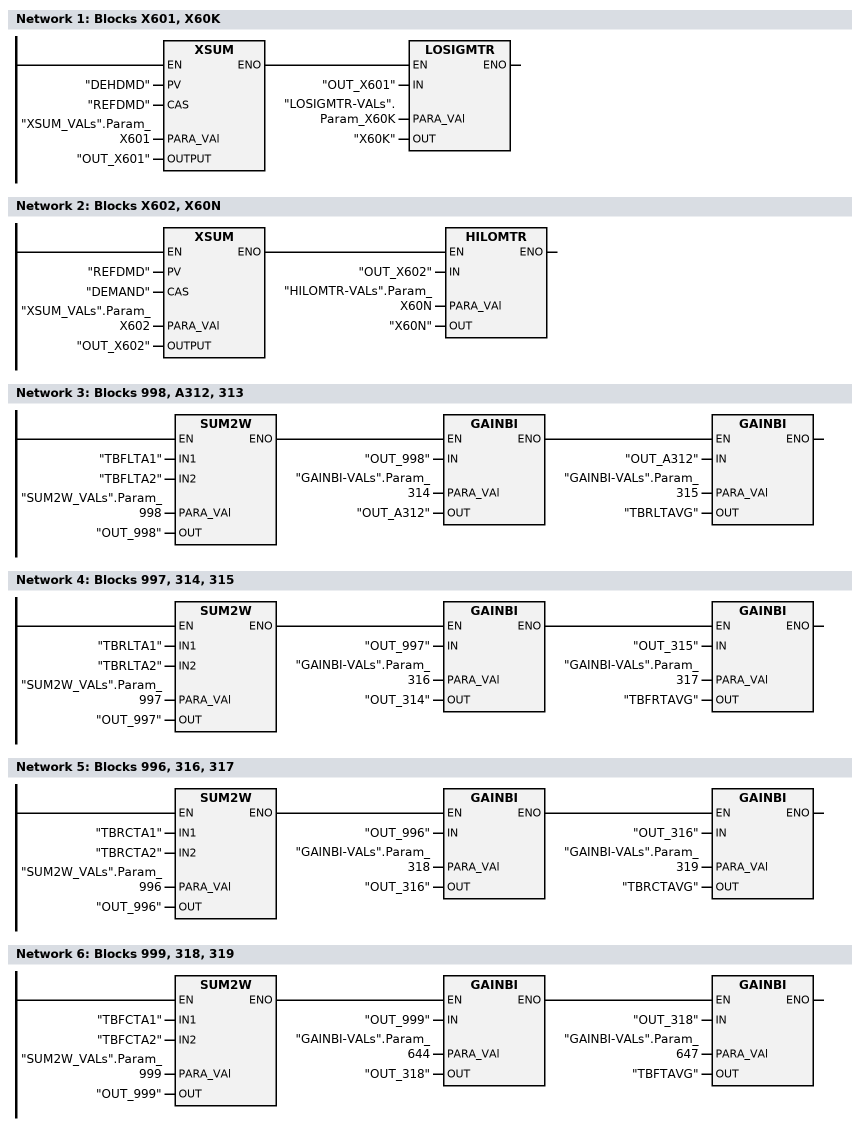
NETWORK
TITLE = Blocks X601, X60K
      A(;
      CALL  "XSUM" (
           PV                       := "DEHDMD",
           CAS                      := "REFDMD",
           PARA_VAl                 := "XSUM_VALs".Param_X601,
           OUTPUT                   := "OUT_X601");
      A     BR;
      );
      JNB   _001;
      CALL  "LOSIGMTR" (
           IN                       := "OUT_X601",
           PARA_VAl                 := "LOSIGMTR-VALs".Param_X60K,
           OUT                      := "X60K");
_001: NOP   0;
NETWORK
TITLE = Blocks X602, X60N
      A(;
      CALL  "XSUM" (
           PV                       := "REFDMD",
           CAS                      := "DEMAND",
           PARA_VAl                 := "XSUM_VALs".Param_X602,
           OUTPUT                   := "OUT_X602");
      A     BR;
      );
      JNB   _002;
      CALL  "HILOMTR" (
           IN                       := "OUT_X602",
           PARA_VAl                 := "HILOMTR-VALs".Param_X60N,
           OUT                      := "X60N");
_002: NOP   0;
NETWORK
TITLE = Blocks 998, A312, 313
      A(;
      A(;
      CALL  "SUM2W" (
           IN1                      := "TBFLTA1",
           IN2                      := "TBFLTA2",
           PARA_VAl                 := "SUM2W_VALs".Param_998,
           OUT                      := "OUT_998");
      A     BR;
      );
      JNB   _003;
      CALL  "GAINBI" (
           IN                       := "OUT_998",
           PARA_VAl                 := "GAINBI-VALs".Param_314,
           OUT                      := "OUT_A312");
_003: A     BR;
      );
      JNB   _004;
      CALL  "GAINBI" (
           IN                       := "OUT_A312",
           PARA_VAl                 := "GAINBI-VALs".Param_315,
           OUT                      := "TBRLTAVG");
_004: NOP   0;
NETWORK
TITLE = Blocks 997, 314, 315
      A(;
      A(;
      CALL  "SUM2W" (
           IN1                      := "TBRLTA1",
           IN2                      := "TBRLTA2",
           PARA_VAl                 := "SUM2W_VALs".Param_997,
           OUT                      := "OUT_997");
      A     BR;
      );
      JNB   _005;
      CALL  "GAINBI" (
           IN                       := "OUT_997",
           PARA_VAl                 := "GAINBI-VALs".Param_316,
           OUT                      := "OUT_314");
_005: A     BR;
      );
      JNB   _006;
      CALL  "GAINBI" (
           IN                       := "OUT_315",
           PARA_VAl                 := "GAINBI-VALs".Param_317,
           OUT                      := "TBFRTAVG");
_006: NOP   0;
NETWORK
TITLE = Blocks 996, 316, 317
      A(;
      A(;
      CALL  "SUM2W" (
           IN1                      := "TBRCTA1",
           IN2                      := "TBRCTA2",
           PARA_VAl                 := "SUM2W_VALs".Param_996,
           OUT                      := "OUT_996");
      A     BR;
      );
      JNB   _007;
      CALL  "GAINBI" (
           IN                       := "OUT_996",
           PARA_VAl                 := "GAINBI-VALs".Param_318,
           OUT                      := "OUT_316");
_007: A     BR;
      );
      JNB   _008;
      CALL  "GAINBI" (
           IN                       := "OUT_316",
           PARA_VAl                 := "GAINBI-VALs".Param_319,
           OUT                      := "TBRCTAVG");
_008: NOP   0;
NETWORK
TITLE = Blocks 999, 318, 319
      A(;
      A(;
      CALL  "SUM2W" (
           IN1                      := "TBFCTA1",
           IN2                      := "TBFCTA2",
           PARA_VAl                 := "SUM2W_VALs".Param_999,
           OUT                      := "OUT_999");
      A     BR;
      );
      JNB   _009;
      CALL  "GAINBI" (
           IN                       := "OUT_999",
           PARA_VAl                 := "GAINBI-VALs".Param_644,
           OUT                      := "OUT_318");
_009: A     BR;
      );
      JNB   _00a;
      CALL  "GAINBI" (
           IN                       := "OUT_318",
           PARA_VAl                 := "GAINBI-VALs".Param_647,
           OUT                      := "TBFTAVG");
_00a: NOP   0;
NETWORK
TITLE = Blocks AIN, 311, X222, X22M
      A(;
      A     "X01I";
      =     L 0.0;
      BLD   103;
      A(;
      A(;
      CALL  "AIN" , "AIN_VALs_POS_2" (
           IN                       := "ROTECC_W",
           OUT                      := "ROTECC");
      A     BR;
      );
      JNB   _00b;
      CALL  "GAINBI" (
           IN                       := "ROTECC",
           PARA_VAl                 := "GAINBI-VALs".Param_313,
           OUT                      := "ROTECCE");
_00b: A     BR;
      );
      JNB   _00c;
      CALL  "TRANSF" (
           FLAG                     := L 0.0,
           IN1_y                    := "A50",
           IN2_n                    := "ROTECCE",
           OUT                      := "OUT_X222");
_00c: A     BR;
      );
      JNB   _00d;
      CALL  "HISIGMTR" (
           IN                       := "OUT_X222",
           PARA_VAl                 := "HISIGMTR-VALs".Param_926,
           OUT                      := "X22M");
_00d: NOP   0;
END_FUNCTION

FUNCTION "Sheet 36 (ATC)" : VOID	// FC 121
TITLE = Sheet 36 (ATC)
//LADDERS 27, 600. ATC PLATEAU FLAGS (Digital)
AUTHOR : RJ
FAMILY : ATC
VERSION : 0.1
BEGIN
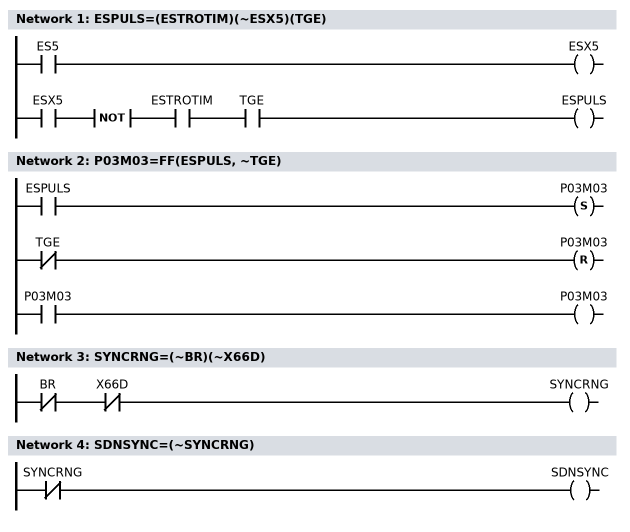
NETWORK
TITLE = ESPULS=(ESTROTIM)(~ESX5)(TGE)
//ESX5=ES5
//
      A     "ES5";
      =     "ESX5";
      A     "ESX5";
      NOT;
      A     "ESTROTIM";
      A     "TGE";
      =     "ESPULS";
NETWORK
TITLE = P03M03=FF(ESPULS, ~TGE)
      A     "ESPULS";
      S     "P03M03";
      AN    "TGE";
      R     "P03M03";
      A     "P03M03";
      =     "P03M03";
NETWORK
TITLE = SYNCRNG=(~BR)(~X66D)
      AN    "BR";
      AN    "X66D";
      =     "SYNCRNG";
NETWORK
TITLE = SDNSYNC=(~SYNCRNG)
      AN    "SYNCRNG";
      =     "SDNSYNC";
END_FUNCTION

FUNCTION "Sheet 37 (ATC)" : VOID	// FC 122
TITLE = Sheet 37 (ATC)
//OVERRIDE LOGIC (Analog)
AUTHOR : RJ
FAMILY : ATC
VERSION : 0.1
BEGIN
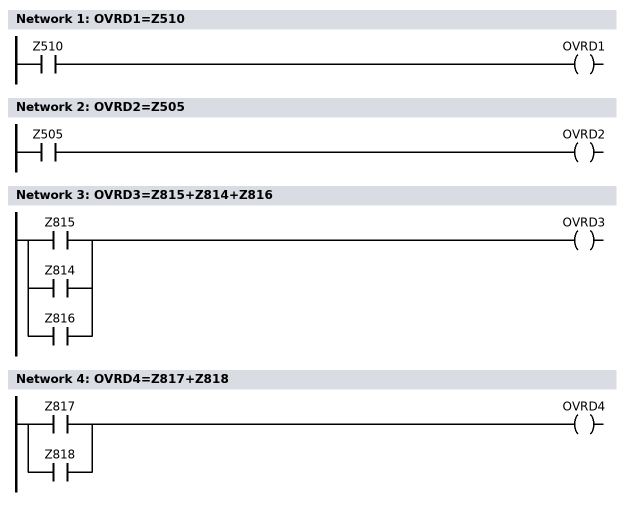
NETWORK
TITLE = OVRD1=Z510
      A     "Z510";
      =     "OVRD1";
NETWORK
TITLE = OVRD2=Z505
      A     "Z505";
      =     "OVRD2";
NETWORK
TITLE = OVRD3=Z815+Z814+Z816
      O     "Z815";
      O     "Z814";
      O     "Z816";
      =     "OVRD3";
NETWORK
TITLE = OVRD4=Z817+Z818
      O     "Z817";
      O     "Z818";
      =     "OVRD4";
END_FUNCTION

FUNCTION "Sheet 38 (ATC)" : VOID	// FC 123
TITLE = Sheet 38 (ATC)
//OVERRIDE LOGIC (Digital)
AUTHOR : RJ
FAMILY : ATC
VERSION : 0.1
BEGIN
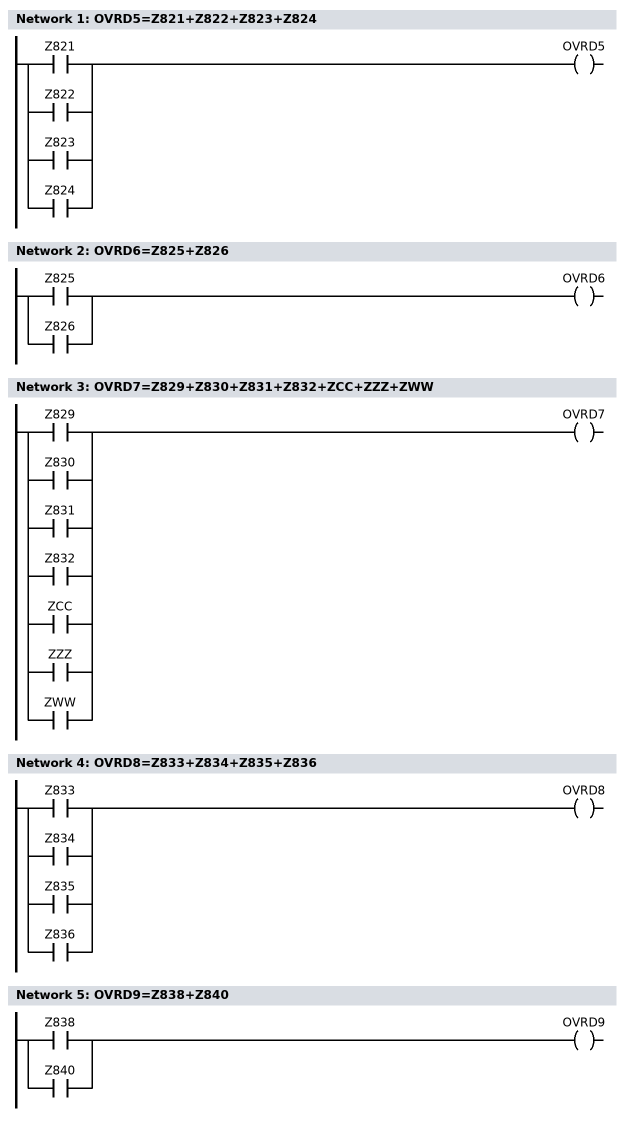
NETWORK
TITLE = OVRD5=Z821+Z822+Z823+Z824
      O     "Z821";
      O     "Z822";
      O     "Z823";
      O     "Z824";
      =     "OVRD5";
NETWORK
TITLE = OVRD6=Z825+Z826
      O     "Z825";
      O     "Z826";
      =     "OVRD6";
NETWORK
TITLE = OVRD7=Z829+Z830+Z831+Z832+ZCC+ZZZ+ZWW
      O     "Z829";
      O     "Z830";
      O     "Z831";
      O     "Z832";
      O     "ZCC";
      O     "ZZZ";
      O     "ZWW";
      =     "OVRD7";
NETWORK
TITLE = OVRD8=Z833+Z834+Z835+Z836
      O     "Z833";
      O     "Z834";
      O     "Z835";
      O     "Z836";
      =     "OVRD8";
NETWORK
TITLE = OVRD9=Z838+Z840
      O     "Z838";
      O     "Z840";
      =     "OVRD9";
END_FUNCTION

FUNCTION "Sheet 39 (ATC)" : VOID	// FC 124
TITLE = Sheet 39 (ATC)
//OVERRIDE LOGIC (Digital)
AUTHOR : RJ
FAMILY : ATC
VERSION : 0.1
BEGIN
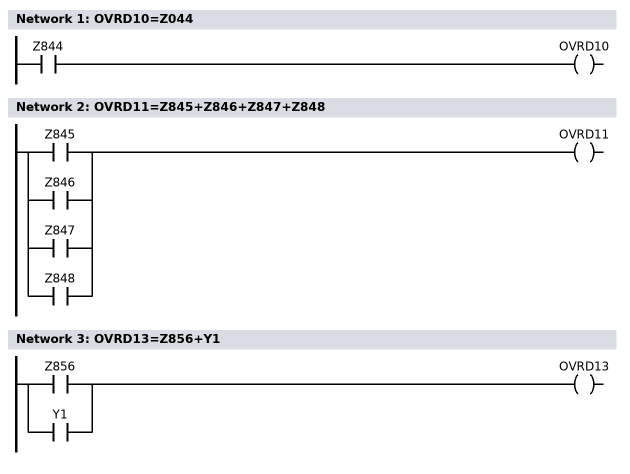
NETWORK
TITLE = OVRD10=Z044
      A     "Z844";
      =     "OVRD10";
NETWORK
TITLE = OVRD11=Z845+Z846+Z847+Z848
      O     "Z845";
      O     "Z846";
      O     "Z847";
      O     "Z848";
      =     "OVRD11";
NETWORK
TITLE = OVRD13=Z856+Y1
      O     "Z856";
      O     "Y1";
      =     "OVRD13";
END_FUNCTION

FUNCTION "Sheet 40 (ATC)" : VOID	// FC 125
TITLE = Sheet 40 (ATC)
//LADDERS 200, 201, 203, 220. REQUEST TRIP P07MXX (Digital)
AUTHOR : RJ
FAMILY : ATC
VERSION : 0.1
BEGIN
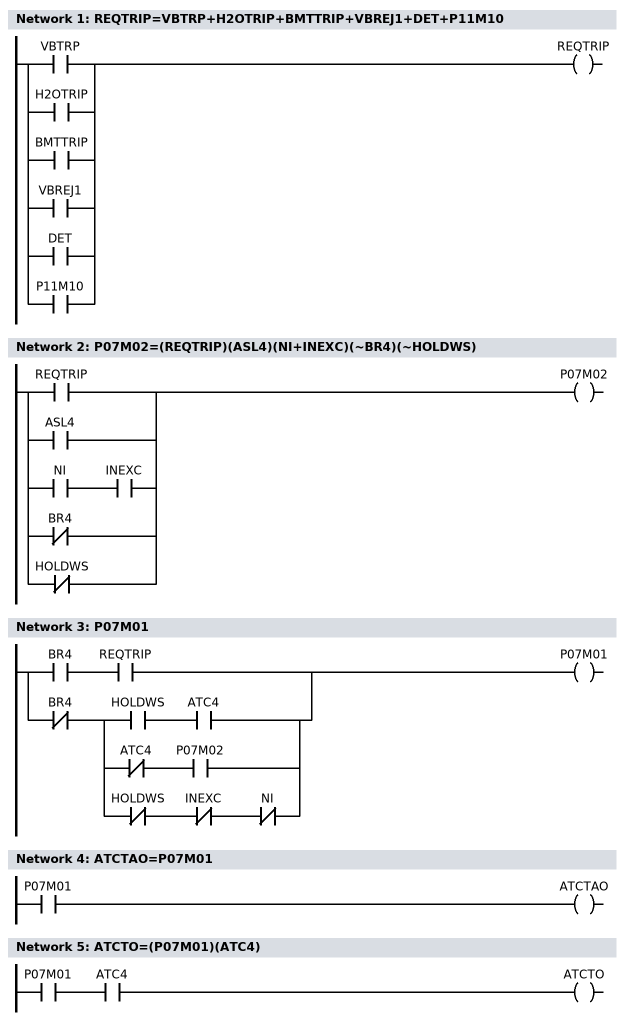
NETWORK
TITLE = REQTRIP=VBTRP+H2OTRIP+BMTTRIP+VBREJ1+DET+P11M10
      O     "VBTRP";
      O     "H2OTRIP";
      O     "BMTTRIP";
      O     "VBREJ1";
      O     "DET";
      O     "P11M10";
      =     "REQTRIP";
NETWORK
TITLE = P07M02=(REQTRIP)(ASL4)(NI+INEXC)(~BR4)(~HOLDWS)
      O     "REQTRIP";
      O     "ASL4";
      O;
      A     "NI";
      A     "INEXC";
      ON    "BR4";
      ON    "HOLDWS";
      =     "P07M02";
NETWORK
TITLE = P07M01
//P07M01=[(BR4)(REQTRIP)]+[(~BR4){(HOLDWS)(ATC4)+(~ATC4)(P07M02)+(~HOLDWS)
//(~INEXC)(~NI)}]
      A     "BR4";
      A     "REQTRIP";
      O;
      AN    "BR4";
      A(;
      A     "HOLDWS";
      A     "ATC4";
      O;
      AN    "ATC4";
      A     "P07M02";
      O;
      AN    "HOLDWS";
      AN    "INEXC";
      AN    "NI";
      );
      =     "P07M01";
NETWORK
TITLE = ATCTAO=P07M01
      A     "P07M01";
      =     "ATCTAO";
NETWORK
TITLE = ATCTO=(P07M01)(ATC4)
      A     "P07M01";
      A     "ATC4";
      =     "ATCTO";
END_FUNCTION

FUNCTION "Sheet 41 (ATC)" : VOID	// FC 126
TITLE = Sheet 41 (ATC)
//LADDERS 201, 202, 203. HOLD 1 & 2 - P07M13 (Digital)
AUTHOR : RJ
FAMILY : ATC
VERSION : 0.1
BEGIN
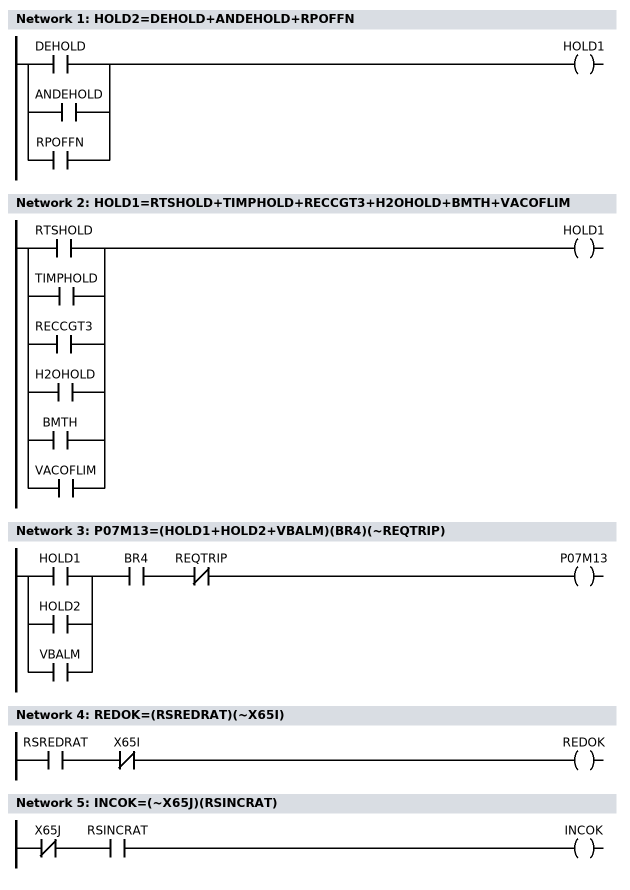
NETWORK
TITLE = HOLD2=DEHOLD+ANDEHOLD+RPOFFN
      O     "DEHOLD";
      O     "ANDEHOLD";
      O     "RPOFFN";
      =     "HOLD1";
NETWORK
TITLE = HOLD1=RTSHOLD+TIMPHOLD+RECCGT3+H2OHOLD+BMTH+VACOFLIM
      O     "RTSHOLD";
      O     "TIMPHOLD";
      O     "RECCGT3";
      O     "H2OHOLD";
      O     "BMTH";
      O     "VACOFLIM";
      =     "HOLD1";
NETWORK
TITLE = P07M13=(HOLD1+HOLD2+VBALM)(BR4)(~REQTRIP)
      A(;
      O     "HOLD1";
      O     "HOLD2";
      O     "VBALM";
      );
      A     "BR4";
      AN    "REQTRIP";
      =     "P07M13";
NETWORK
TITLE = REDOK=(RSREDRAT)(~X65I)
      A     "RSREDRAT";
      AN    "X65I";
      =     "REDOK";
NETWORK
TITLE = INCOK=(~X65J)(RSINCRAT)
      AN    "X65J";
      A     "RSINCRAT";
      =     "INCOK";
END_FUNCTION

FUNCTION "Sheet 42 (ATC)" : VOID	// FC 127
TITLE = Sheet 42 (ATC)
//LADDERS 110, 111, 112, 113. OVERRIDE & P07M12 (Digital)
AUTHOR : RJ
FAMILY : ATC
VERSION : 0.1
BEGIN
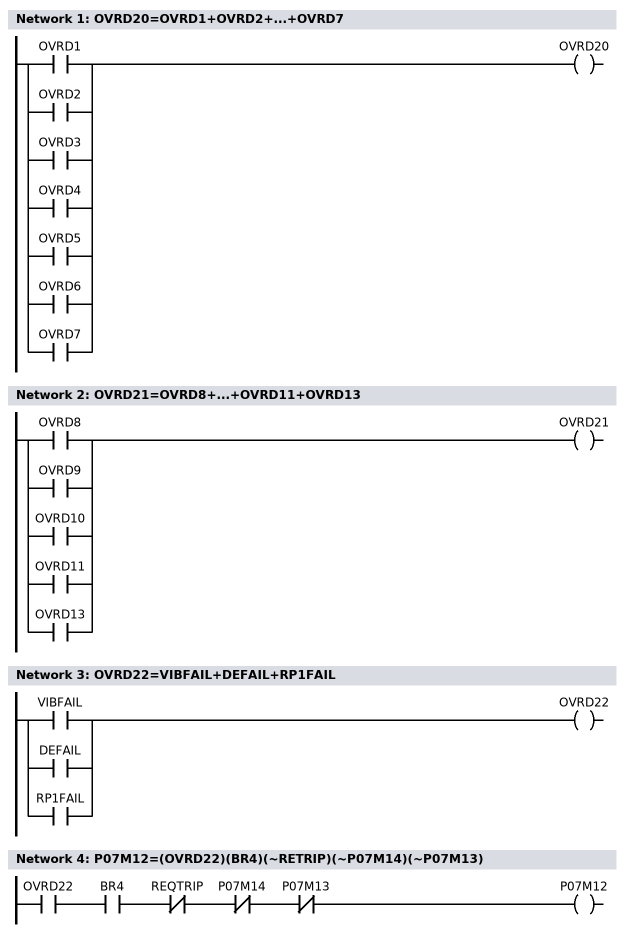
NETWORK
TITLE = OVRD20=OVRD1+OVRD2+...+OVRD7
      O     "OVRD1";
      O     "OVRD2";
      O     "OVRD3";
      O     "OVRD4";
      O     "OVRD5";
      O     "OVRD6";
      O     "OVRD7";
      =     "OVRD20";
NETWORK
TITLE = OVRD21=OVRD8+...+OVRD11+OVRD13
      O     "OVRD8";
      O     "OVRD9";
      O     "OVRD10";
      O     "OVRD11";
      O     "OVRD13";
      =     "OVRD21";
NETWORK
TITLE = OVRD22=VIBFAIL+DEFAIL+RP1FAIL
      O     "VIBFAIL";
      O     "DEFAIL";
      O     "RP1FAIL";
      =     "OVRD22";
NETWORK
TITLE = P07M12=(OVRD22)(BR4)(~RETRIP)(~P07M14)(~P07M13)
      A     "OVRD22";
      A     "BR4";
      AN    "REQTRIP";
      AN    "P07M14";
      AN    "P07M13";
      =     "P07M12";
END_FUNCTION

FUNCTION "Sheet 43 (ATC)" : VOID	// FC 128
TITLE = Sheet 43 (ATC)
//LADDERS 11, 113, 114. HOLD LOAD & P07M09 - 14 (Digital)
AUTHOR : RJ
FAMILY : ATC
VERSION : 0.1
BEGIN
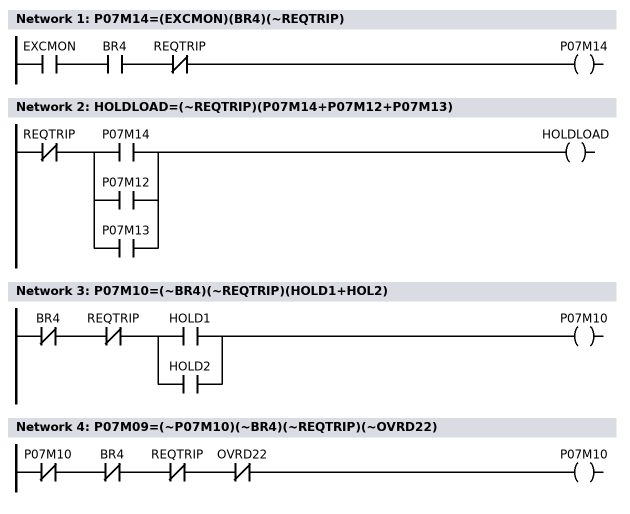
NETWORK
TITLE = P07M14=(EXCMON)(BR4)(~REQTRIP)
      A     "EXCMON";
      A     "BR4";
      AN    "REQTRIP";
      =     "P07M14";
NETWORK
TITLE = HOLDLOAD=(~REQTRIP)(P07M14+P07M12+P07M13)
      AN    "REQTRIP";
      A(;
      O     "P07M14";
      O     "P07M12";
      O     "P07M13";
      );
      =     "HOLDLOAD";
NETWORK
TITLE = P07M10=(~BR4)(~REQTRIP)(HOLD1+HOL2)
      AN    "BR4";
      AN    "REQTRIP";
      A(;
      O     "HOLD1";
      O     "HOLD2";
      );
      =     "P07M10";
NETWORK
TITLE = P07M09=(~P07M10)(~BR4)(~REQTRIP)(~OVRD22)
      AN    "P07M10";
      AN    "BR4";
      AN    "REQTRIP";
      AN    "OVRD22";
      =     "P07M10";
END_FUNCTION

FUNCTION "Sheet 44 (ATC)" : VOID	// FC 129
TITLE = Sheet 44 (ATC)
//LADDERS 115, 116. HOLD WS & P07M02 - 04 (Digital)
AUTHOR : RJ
FAMILY : ATC
VERSION : 0.1
BEGIN
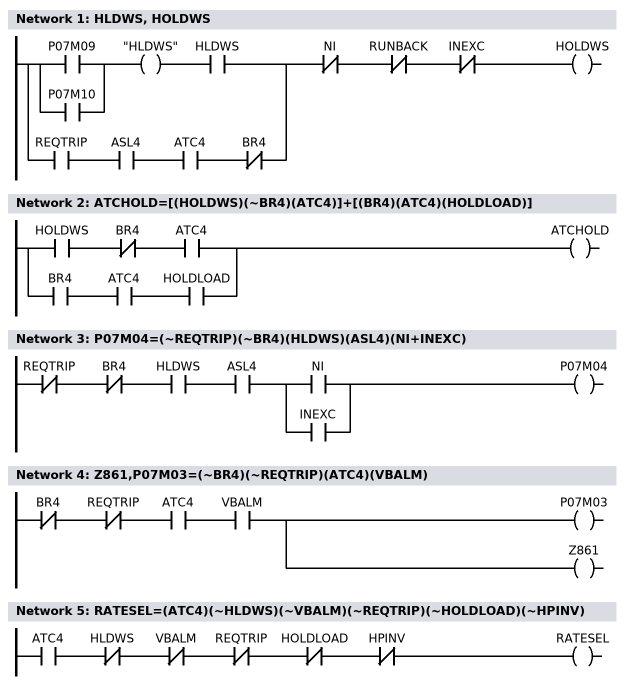
NETWORK
TITLE = HLDWS, HOLDWS
//HOLDWS={HLDWS+(REQTRIP)(ASL4)(ATC4)(~BR4)}{~NI}{~RUNBACK}{~INEXC}
//HLDWS=P07M09+P07M10
      A(;
      A(;
      O     "P07M09";
      O     "P07M10";
      );
      =     "HLDWS";
      A     "HLDWS";
      O;
      A     "REQTRIP";
      A     "ASL4";
      A     "ATC4";
      AN    "BR4";
      );
      AN    "NI";
      AN    "RUNBACK";
      AN    "INEXC";
      =     "HOLDWS";
NETWORK
TITLE = ATCHOLD=[(HOLDWS)(~BR4)(ATC4)]+[(BR4)(ATC4)(HOLDLOAD)]
      A     "HOLDWS";
      AN    "BR4";
      A     "ATC4";
      O;
      A     "BR4";
      A     "ATC4";
      A     "HOLDLOAD";
      =     "ATCHOLD";
NETWORK
TITLE = P07M04=(~REQTRIP)(~BR4)(HLDWS)(ASL4)(NI+INEXC)
      AN    "REQTRIP";
      AN    "BR4";
      A     "HLDWS";
      A     "ASL4";
      A(;
      O     "NI";
      O     "INEXC";
      );
      =     "P07M04";
NETWORK
TITLE = Z861,P07M03=(~BR4)(~REQTRIP)(ATC4)(VBALM)
      AN    "BR4";
      AN    "REQTRIP";
      A     "ATC4";
      A     "VBALM";
      =     "P07M03";
      =     "Z861";
NETWORK
TITLE = RATESEL=(ATC4)(~HLDWS)(~VBALM)(~REQTRIP)(~HOLDLOAD)(~HPINV)
      A     "ATC4";
      AN    "HLDWS";
      AN    "VBALM";
      AN    "REQTRIP";
      AN    "HOLDLOAD";
      AN    "HPINV";
      =     "RATESEL";
END_FUNCTION

FUNCTION "Sheet 45 (ATC)" : VOID	// FC 130
TITLE = Sheet 45 (ATC)
//LADDERS 117, 118. LOAD RATE INC/DEC P07M05 - 08 (Digital)
AUTHOR : RJ
FAMILY : ATC
VERSION : 0.1
BEGIN
NETWORK
TITLE = MOVERATE=(RATETIME)(~SAMERATE)
//RATETIME=FF[ON{(RATESEL)(~RATETIME)},RATETIME]
      A(;
      A(;
      A     "RATESEL";
      AN    "RATETIME";
      L     "ATCTime_VALs".T10ON;
      SD    T 10;
      NOP   0;
      NOP   0;
      NOP   0;
      A     T 10;
      );
      S     "RATETIME";
      A     "RATETIME";
      R     "RATETIME";
      A     "RATETIME";
      );
      =     "RATETIME";
      A     "RATETIME";
      AN    "SAMERATE";
      =     "MOVERATE";
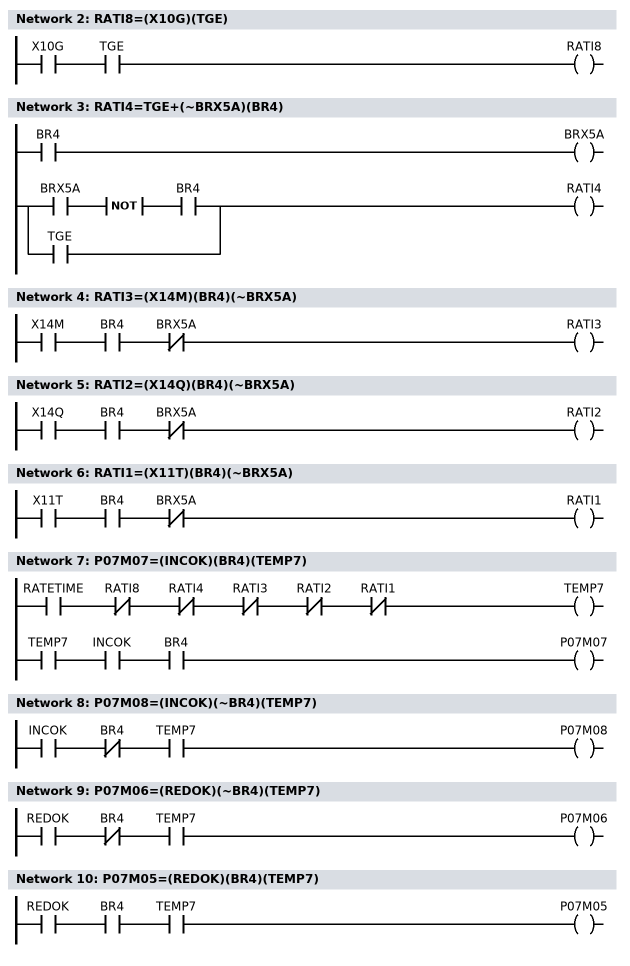
NETWORK
TITLE = RATI8=(X10G)(TGE)
      A     "X10G";
      A     "TGE";
      =     "RATI8";
NETWORK
TITLE = RATI4=TGE+(~BRX5A)(BR4)
//BRX5A=BR4
//
      A     "BR4";
      =     "BRX5A";
      A     "BRX5A";
      NOT;
      A     "BR4";
      O     "TGE";
      =     "RATI4";
NETWORK
TITLE = RATI3=(X14M)(BR4)(~BRX5A)
      A     "X14M";
      A     "BR4";
      AN    "BRX5A";
      =     "RATI3";
NETWORK
TITLE = RATI2=(X14Q)(BR4)(~BRX5A)
      A     "X14Q";
      A     "BR4";
      AN    "BRX5A";
      =     "RATI2";
NETWORK
TITLE = RATI1=(X11T)(BR4)(~BRX5A)
      A     "X11T";
      A     "BR4";
      AN    "BRX5A";
      =     "RATI1";
NETWORK
TITLE = P07M07=(INCOK)(BR4)(TEMP7)
//TEMP7=(RATETIME)(~RATI8)(~RATI4)(~RATI3)(~RATI2)(~RATI1)
      A     "RATETIME";
      AN    "RATI8";
      AN    "RATI4";
      AN    "RATI3";
      AN    "RATI2";
      AN    "RATI1";
      =     "TEMP7";
      A     "TEMP7";
      A     "INCOK";
      A     "BR4";
      =     "P07M07";
NETWORK
TITLE = P07M08=(INCOK)(~BR4)(TEMP7)
      A     "INCOK";
      AN    "BR4";
      A     "TEMP7";
      =     "P07M08";
NETWORK
TITLE = P07M06=(REDOK)(~BR4)(TEMP7)
      A     "REDOK";
      AN    "BR4";
      A     "TEMP7";
      =     "P07M06";
NETWORK
TITLE = P07M05=(REDOK)(BR4)(TEMP7)
      A     "REDOK";
      A     "BR4";
      A     "TEMP7";
      =     "P07M05";
END_FUNCTION

FUNCTION "Sheet 47 (ATC)" : VOID	// FC 131
TITLE = Sheet 47 (ATC)
//LADDERS 118, 192. P00M00A-G (Digital)
AUTHOR : RJ
FAMILY : ATC
VERSION : 0.1
BEGIN
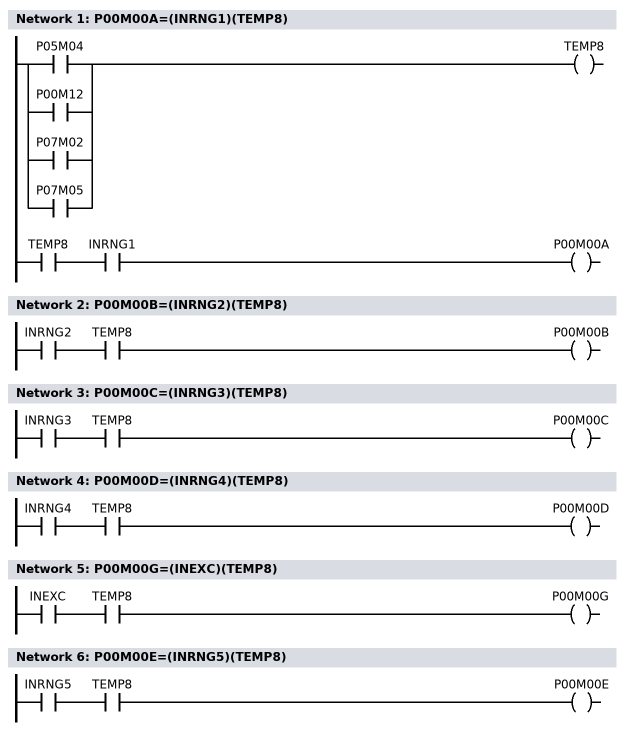
NETWORK
TITLE = P00M00A=(INRNG1)(TEMP8)
//TEMP8=P05M04+P00M12+P07M02+P07M04
//
      A(;
      O     "P05M04";
      O     "P00M12";
      O     "P07M02";
      O     "P07M05";
      );
      =     "TEMP8";
      A     "TEMP8";
      A     "INRNG1";
      =     "P00M00A";
NETWORK
TITLE = P00M00B=(INRNG2)(TEMP8)
      A     "INRNG2";
      A     "TEMP8";
      =     "P00M00B";
NETWORK
TITLE = P00M00C=(INRNG3)(TEMP8)
      A     "INRNG3";
      A     "TEMP8";
      =     "P00M00C";
NETWORK
TITLE = P00M00D=(INRNG4)(TEMP8)
      A     "INRNG4";
      A     "TEMP8";
      =     "P00M00D";
NETWORK
TITLE = P00M00G=(INEXC)(TEMP8)
      A     "INEXC";
      A     "TEMP8";
      =     "P00M00G";
NETWORK
TITLE = P00M00E=(INRNG5)(TEMP8)
      A     "INRNG5";
      A     "TEMP8";
      =     "P00M00E";
END_FUNCTION

FUNCTION "Sheet 46 (ATC)" : VOID	// FC 132
TITLE = Sheet 46 (ATC)
//LOOPS 63, 65. LOAD RATE (Analog)
AUTHOR : RJ
FAMILY : ATC
VERSION : 0.1
BEGIN
NETWORK
TITLE = Blocks X652, X654
      A     "MOVERATE";
      =     L 0.0;
      BLD   103;
      A(;
      A     "RSINCRAT";
      =     L 0.1;
      BLD   103;
      CALL  "XTRANSF" (
           PV_Y                     := "Constants_RSM".A40,
           CAS_N                    := "Constants_RSM".A40,
           FLAG                     := L 0.1,
           PARA_VAl                 := "XTRANSF_VALs".Param_X652,
           OUTPUT                   := "OUT_X652");
      A     BR;
      );
      JNB   _001;
      CALL  "XTRANSF" (
           PV_Y                     := "OUT_X652",
           CAS_N                    := "Constants_RSM".A40,
           FLAG                     := L 0.0,
           PARA_VAl                 := "XTRANSF_VALs".Param_X654,
           OUTPUT                   := "OUT_X654");
_001: NOP   0;
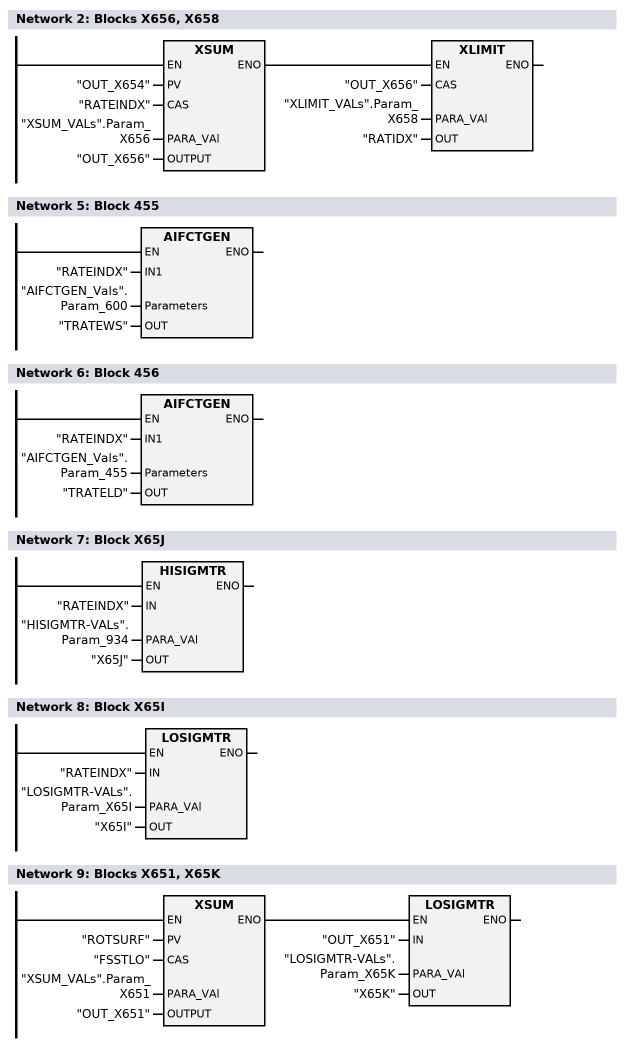
NETWORK
TITLE = Blocks X656, X658
      A(;
      CALL  "XSUM" (
           PV                       := "OUT_X654",
           CAS                      := "RATEINDX",
           PARA_VAl                 := "XSUM_VALs".Param_X656,
           OUTPUT                   := "OUT_X656");
      A     BR;
      );
      JNB   _002;
      CALL  "XLIMIT" (
           CAS                      := "OUT_X656",
           PARA_VAl                 := "XLIMIT_VALs".Param_X658,
           OUT                      := "RATIDX");
_002: NOP   0;
NETWORK
TITLE = Blocks X631, X633, X635
      A     "RATI2";
      =     L 0.0;
      BLD   103;
      A(;
      A     "RATI3";
      =     L 0.1;
      BLD   103;
      A(;
      A     "RATI4";
      =     L 0.2;
      BLD   103;
      CALL  "XTRANSF" (
           PV_Y                     := "Constants_RSM".A40,
           CAS_N                    := "RATIDX",
           FLAG                     := L 0.2,
           PARA_VAl                 := "XTRANSF_VALs".Param_X631,
           OUTPUT                   := "OUT_X631");
      A     BR;
      );
      JNB   _003;
      CALL  "XTRANSF" (
           PV_Y                     := "Constants_RSM".A40,
           CAS_N                    := "OUT_X631",
           FLAG                     := L 0.1,
           PARA_VAl                 := "XTRANSF_VALs".Param_X633,
           OUTPUT                   := "OUT_X633");
_003: A     BR;
      );
      JNB   _004;
      CALL  "XTRANSF" (
           PV_Y                     := "Constants_RSM".A40,
           CAS_N                    := "OUT_X633",
           FLAG                     := L 0.0,
           PARA_VAl                 := "XTRANSF_VALs".Param_X635,
           OUTPUT                   := "OUT_X635");
_004: NOP   0;
NETWORK
TITLE = Blocks X637, X638, XA638
      A(;
      A     "RATI8";
      =     L 0.0;
      BLD   103;
      A(;
      A     "RATI1";
      =     L 0.1;
      BLD   103;
      CALL  "XTRANSF" (
           PV_Y                     := "Constants_RSM".A40,
           CAS_N                    := "OUT_X635",
           FLAG                     := L 0.1,
           PARA_VAl                 := "XTRANSF_VALs".Param_X637,
           OUTPUT                   := "RATETEMP");
      A     BR;
      );
      JNB   _005;
      CALL  "XTRANSF" (
           PV_Y                     := "Constants_RSM".A40,
           CAS_N                    := "RATETEMP",
           FLAG                     := L 0.0,
           PARA_VAl                 := "XTRANSF_VALs".Param_X638,
           OUTPUT                   := "OUT_X638");
_005: A     BR;
      );
      JNB   _006;
      CALL  "XLIMIT" (
           CAS                      := "OUT_X638",
           PARA_VAl                 := "XLIMIT_VALs".Param_XA638,
           OUT                      := "RATEINDX");
_006: NOP   0;
NETWORK
TITLE = Block 455
      CALL  "AIFCTGEN" (
           IN1                      := "RATEINDX",
           Parameters               := "AIFCTGEN_Vals".Param_600,
           OUT                      := "TRATEWS");
      NOP   0;
NETWORK
TITLE = Block 456
      CALL  "AIFCTGEN" (
           IN1                      := "RATEINDX",
           Parameters               := "AIFCTGEN_Vals".Param_455,
           OUT                      := "TRATELD");
      NOP   0;
NETWORK
TITLE = Block X65J
      CALL  "HISIGMTR" (
           IN                       := "RATEINDX",
           PARA_VAl                 := "HISIGMTR-VALs".Param_934,
           OUT                      := "X65J");
      NOP   0;
NETWORK
TITLE = Block X65I
      CALL  "LOSIGMTR" (
           IN                       := "RATEINDX",
           PARA_VAl                 := "LOSIGMTR-VALs".Param_X65I,
           OUT                      := "X65I");
      NOP   0;
NETWORK
TITLE = Blocks X651, X65K
      A(;
      CALL  "XSUM" (
           PV                       := "ROTSURF",
           CAS                      := "FSSTLO",
           PARA_VAl                 := "XSUM_VALs".Param_X651,
           OUTPUT                   := "OUT_X651");
      A     BR;
      );
      JNB   _007;
      CALL  "LOSIGMTR" (
           IN                       := "OUT_X651",
           PARA_VAl                 := "LOSIGMTR-VALs".Param_X65K,
           OUT                      := "X65K");
_007: NOP   0;
END_FUNCTION

FUNCTION "Sheet 48_49 (ATC)" : VOID	// FC 133
TITLE = Sheet 48_49 (ATC)
//
//Initialization of ATC constants from AVALGEN DB
//
AUTHOR : RJ
FAMILY : ATC
VERSION : 0.0
BEGIN
// body was compiled from an SCL source; compiled code not shown
END_FUNCTION

DATA_BLOCK "Constants_RSM"	// DB 1
AUTHOR : RJ
FAMILY : RSM
VERSION : 0.1
  STRUCT
   A40 : REAL ;	//Sheet 2 (RSM)
   KELVIN : REAL  := 4.600000e+002;	//Sheet 2 (RSM)
   AV1 : REAL  := 1.000000e+000;	//Sheet 2 (RSM)
   C12STR : REAL  := -3.862000e-005;	//=C12 Value. Sheet 2 (RSM)
   C11STR : REAL ;	//=C11 Value. Sheet 2 (RSM)
   C10STR : REAL ;	//=C10 Value. Sheet 2 (RSM)
   C31 : REAL  := 8.617000e-001;	//Sheet 2 (RSM)
   C11 : REAL  := 2.800000e-004;	//Sheet 2 (RSM)
   HOTDIFLM : REAL  := 7.326000e+001;	//Sheet 2 (RSM)
   GLRATE : REAL  := 1.625000e+001;	//=LRATE(10). Sheet 2 (RSM)
   TDEM : REAL  := 7.166000e+000;	//Sheet 2 (RSM)
   C1 : REAL ;	//Sheet 2 (RSM)
   C2 : REAL ;	//Sheet 2 (RSM)
   C3 : REAL ;	//Sheet 2 (RSM)
   C4 : REAL ;	//Sheet 2 (RSM)
   C5 : REAL ;	//Sheet 2 (RSM)
   C6 : REAL  := 1.500000e+003;	//Sheet 2 (RSM)
   C7 : REAL ;	//Sheet 2 (RSM)
   C8 : REAL ;	//Sheet 2 (RSM)
   C9 : REAL ;	//Sheet 2 (RSM)
   C10 : REAL ;	//Sheet 2 (RSM)
   C12 : REAL  := -3.862000e-005;	//Sheet 2 (RSM)
   C13 : REAL ;	//Sheet 2 (RSM)
   C14 : REAL ;	//Sheet 2 (RSM)
   C15 : REAL ;	//Sheet 2 (RSM)
   C16 : REAL ;	//Sheet 2 (RSM)
   C17 : REAL ;	//Sheet 2 (RSM)
   C18 : REAL ;	//Sheet 2 (RSM)
   C19 : REAL ;	//Sheet 2 (RSM)
   C20 : REAL ;	//Sheet 2 (RSM)
   C21 : REAL ;	//Sheet 2 (RSM)
   C22 : REAL ;	//Sheet 2 (RSM)
   C23 : REAL ;	//Sheet 2 (RSM)
   C24 : REAL ;	//Sheet 2 (RSM)
   C25 : REAL ;	//Sheet 2 (RSM)
   C26 : REAL ;	//Sheet 2 (RSM)
   C27 : REAL ;	//Sheet 2 (RSM)
   N300 : REAL ;	//Sheet 2 (RSM)
   MWRATED : REAL  := 3.250000e+002;	//Unit MW rating. Sheet 2 (RSM)
   DVTRUE : BOOL  := TRUE;	//Sheet 2 (RSM)
   DVFALSE : BOOL ;	//Sheet 2 (RSM)
   DX1PASS : BOOL ;	//=TRUE for the first loop time only after drop power up or reset. Sheet 2 (RSM)
   NDIFLM : REAL  := 7.326000e+001;	//Sheet 2 (RSM)
   FSST : REAL ;	//Sheet 20 (RSM)
  END_STRUCT ;	
BEGIN
   KELVIN := 4.600000e+02;
   AV1 := 1.000000e+00;
   DVTRUE := TRUE;
END_DATA_BLOCK

DATA_BLOCK "HISIGMTR-VALs"	// DB 2
AUTHOR : sabeeh
VERSION : 0.1
  STRUCT
   Param_375 : UDT 1;	//Sheet 3 (RSM)
   Param_X67D : UDT 1;	//Sheet 4 (RSM)
   Param_321 : UDT 1;	//Sheet 4 (RSM)
   Param_320 : UDT 1;	//Sheet 6 (RSM)
   Param_270 : UDT 1;	//Sheet 6 (RSM)
   Param_272 : UDT 1;	//Sheet 6 (RSM)
   Param_318 : UDT 1;	//Sheet 6 (RSM)
   Param_126 : UDT 1;	//Sheet 6 (RSM)
   Param_137 : UDT 1;	//Sheet 8 (RSM)
   Param_221 : UDT 1;	//Sheet 8 (RSM)
   Param_X10G : UDT 1;	//Sheet 11 (RSM)
   Param_X11L : UDT 1;	//Sheet 17 (RSM)
   Param_X73K : UDT 1;	//Sheet 17 (RSM)
   Param_X11P : UDT 1;	//Sheet 17 (RSM)
   Param_X11T : UDT 1;	//Sheet 17 (RSM)
   Param_X11N : UDT 1;	//Sheet 17 (RSM)
   Param_X11R : UDT 1;	//Sheet 17 (RSM)
   Param_X11V : UDT 1;	//Sheet 17 (RSM)
   Param_X09L : UDT 1;	//Sheet 17 (RSM)
   Param_X67A : UDT 1;	//Sheet 17 (RSM)
   Param_X14M : UDT 1;	//Sheet 18 (RSM)
   Param_X14Q : UDT 1;	//Sheet 18 (RSM)
   Param_324 : UDT 1;	//Sheet 21 (RSM)
   Param_X73M : UDT 1;	//Sheet 21 (RSM)
   Param_X30K : UDT 1;	//Sheet 7 (ATC)
   Param_X20B : UDT 1;	//Sheet 11 (ATC)
   Param_X20C : UDT 1;	//Sheet 11 (ATC)
   Param_X20D : UDT 1;	//Sheet 11 (ATC)
   Param_X20E : UDT 1;	//Sheet 11 (ATC)
   Param_X20H : UDT 1;	//Sheet 17 (ATC)
   Param_X41A : UDT 1;	//Sheet 17 (ATC)
   Param_X41B : UDT 1;	//Sheet 17 (ATC)
   Param_806 : UDT 1;	//Sheet 25 (ATC)
   Param_991 : UDT 1;	//Sheet 25 (ATC)
   Param_397 : UDT 1;	//Sheet 25 (ATC)
   Param_X01I : UDT 1;	//Sheet 25 (ATC)
   Param_695 : UDT 1;	//Sheet 30 (ATC)
   Param_X22M : UDT 1;	//Sheet 35 (ATC)
   Param_X65J : UDT 1;	//Sheet 46 (ATC)
   Param_926 : UDT 1;	//Sheet 24 (ATC)
   Param_934 : UDT 1;	//Sheet 24 (ATC)
   Param_942 : UDT 1;	//Sheet 24 (ATC)
   Param_950 : UDT 1;	//Sheet 24 (ATC)
   Param_958 : UDT 1;	//Sheet 24 (ATC)
   Param_966 : UDT 1;	//Sheet 24 (ATC)
   Param_974 : UDT 1;	//Sheet 24 (ATC)
   Param_982 : UDT 1;	//Sheet 24 (ATC)
   Param_890 : UDT 1;	//Sheet 24 (ATC)
   Param_247 : UDT 1;	//Sheet 24 (ATC)
  END_STRUCT ;	
BEGIN
   Param_375.STPT := 1.666700e+01;
   Param_375.DBAN := 1.000000e+00;
   Param_X67D.STPT := 5.100000e+02;
   Param_X67D.DBAN := 2.500000e+00;
   Param_321.STPT := 6.000000e+02;
   Param_321.DBAN := 5.000000e-01;
   Param_320.STPT := 3.000000e+02;
   Param_320.DBAN := 5.000000e-01;
   Param_270.STPT := 1.000000e+00;
   Param_272.STPT := 5.890000e+01;
   Param_318.STPT := 5.000000e+00;
   Param_318.DBAN := 1.000000e-02;
   Param_126.STPT := 6.000000e+01;
   Param_126.DBAN := 5.000000e-01;
   Param_137.STPT := 3.000000e+02;
   Param_221.DBAN := 1.000000e-01;
   Param_X11L.DBAN := 2.000000e-01;
   Param_X73K.DBAN := 5.000000e-01;
   Param_X11P.DBAN := 5.000000e-01;
   Param_X11T.DBAN := 5.000000e-01;
   Param_X11N.DBAN := 1.000000e+00;
   Param_X11R.DBAN := 5.000000e-01;
   Param_X11V.DBAN := 5.000000e-01;
   Param_X67A.STPT := 1.190000e+02;
   Param_X67A.DBAN := 5.000000e-01;
   Param_X14M.DBAN := 5.000000e-01;
   Param_X14Q.DBAN := 5.000000e-01;
   Param_324.STPT := 1.700000e+00;
   Param_324.DBAN := 5.000000e-01;
   Param_X73M.DBAN := 5.000000e-01;
   Param_X30K.STPT := 3.500000e+02;
   Param_X30K.DBAN := 5.000000e+00;
   Param_X20B.STPT := 1.000000e+02;
   Param_X20B.DBAN := 1.000000e+00;
   Param_X20C.STPT := 1.100000e+02;
   Param_X20C.DBAN := 1.000000e+00;
   Param_X20D.STPT := 1.200000e+02;
   Param_X20D.DBAN := 1.000000e+00;
   Param_X20E.STPT := 1.700000e+02;
   Param_X20E.DBAN := 2.000000e+00;
   Param_X20H.STPT := 1.500000e+03;
   Param_X20H.DBAN := 1.000000e+01;
   Param_X41A.STPT := 8.000000e+01;
   Param_X41A.DBAN := 2.000000e+00;
   Param_X41B.STPT := 1.210000e+02;
   Param_X41B.DBAN := 2.000000e+00;
END_DATA_BLOCK

DATA_BLOCK "LOSIGMTR-VALs"	// DB 3
AUTHOR : Sabeeh
VERSION : 0.1
  STRUCT
   Param_130 : UDT 2;	//Sheet 3 (RSM)
   Param_X09K : UDT 2;	//Sheet 17 (RSM)
   Param_325 : UDT 2;	//Sheet 21 (RSM)
   Param_X30L : UDT 2;	//Sheet 7 (ATC)
   Param_X75H : UDT 2;	//Sheet 10 (ATC)
   Param_X75I : UDT 2;	//Sheet 10 (ATC)
   Param_X75J : UDT 2;	//Sheet 10 (ATC)
   Param_X20A : UDT 2;	//Sheet 11 (ATC)
   Param_X41D : UDT 2;	//Sheet 17 (ATC)
   Param_884 : UDT 2;	//Sheet 17 (ATC)
   Param_807 : UDT 2;	//Sheet 25 (ATC)
   Param_992 : UDT 2;	//Sheet 25 (ATC)
   Param_A398 : UDT 2;	//Sheet 25 (ATC)
   Param_696 : UDT 2;	//Sheet 30 (ATC)
   Param_X05G : UDT 2;	//Sheet 33 (ATC)
   Param_X60K : UDT 2;	//Sheet 35 (ATC)
   Param_X65I : UDT 2;	//Sheet 46 (ATC)
   Param_X65K : UDT 2;	//Sheet 46 (ATC)
  END_STRUCT ;	
BEGIN
   Param_130.STPT := 7.200000e+03;
   Param_325.STPT := -1.700000e+00;
   Param_325.DBAN := 5.000000e-01;
   Param_X30L.STPT := 2.500000e+02;
   Param_X30L.DBAN := 5.000000e+00;
   Param_X75H.STPT := 3.000000e+03;
   Param_X75H.DBAN := 5.000000e+00;
   Param_X75I.STPT := 1.000000e+03;
   Param_X75I.DBAN := 5.000000e+00;
   Param_X75J.STPT := 1.350000e+03;
   Param_X75J.DBAN := 5.000000e+00;
   Param_X20A.STPT := 7.000000e+01;
   Param_X20A.DBAN := 1.000000e-01;
   Param_X41D.STPT := 6.000000e+02;
   Param_X41D.DBAN := 5.000000e+00;
   Param_884.DBAN := 1.000000e-01;
END_DATA_BLOCK

DATA_BLOCK "AIN_VALs_VIB"	// DB 4
AUTHOR : RJ
VERSION : 0.1
"AIN"
BEGIN
END_DATA_BLOCK

DATA_BLOCK "GAINBI-VALs"	// DB 5
AUTHOR : Sabeeh
VERSION : 0.1
  STRUCT
   Param_90 : UDT 4;	//Sheet 3 (RSM)
   Param_91 : UDT 4;	//Sheet 3 (RSM)
   Param_057 : UDT 4;	//Sheet 3 (RSM)
   Param_92 : UDT 4;	//Sheet 4 (RSM)
   Param_93 : UDT 4;	//Sheet 4 (RSM)
   Param_88 : UDT 4;	//Sheet 4 (RSM)
   Param_055 : UDT 4;	//Sheet 4 (RSM)
   Param_790 : UDT 4;	//Sheet 4 (RSM)
   Param_224 : UDT 4;	//Sheet 8 (RSM)
   Param_713 : UDT 4;	//Sheet 13 (RSM)
   Param_711 : UDT 4;	//Sheet 13 (RSM)
   Param_294 : UDT 4;	//Sheet 16 (RSM)
   Param_295 : UDT 4;	//Sheet 16 (RSM)
   Param_875 : UDT 4;	//Sheet 20 (RSM)
   Param_143 : UDT 4;	//Sheet 22 (RSM)
   Param_144 : UDT 4;	//Sheet 22 (RSM)
   Param_466 : UDT 4;	//Sheet 37 (RSM)
   Param_468 : UDT 4;	//Sheet 37 (RSM)
   Param_GBA1 : UDT 4;	//Sheet 12 (ATC)
   Param_GBA2 : UDT 4;	//Sheet 12 (ATC)
   Param_GBA3 : UDT 4;	//Sheet 12 (ATC)
   Param_GBA4 : UDT 4;	//Sheet 12 (ATC)
   Param_GBA5 : UDT 4;	//Sheet 12 (ATC)
   Param_GBA6 : UDT 4;	//Sheet 12 (ATC)
   Param_GBA7 : UDT 4;	//Sheet 12 (ATC)
   Param_GBA8 : UDT 4;	//Sheet 12 (ATC)
   Param_GBA9 : UDT 4;	//Sheet 12 (ATC)
   Param_GBA10 : UDT 4;	//Sheet 12 (ATC)
   Param_GBA11 : UDT 4;	//Sheet 12 (ATC)
   Param_GBA12 : UDT 4;	//Sheet 12 (ATC)
   Param_GBA13 : UDT 4;	//Sheet 12 (ATC)
   Param_GBA14 : UDT 4;	//Sheet 12 (ATC)
   Param_GBA15 : UDT 4;	//Sheet 12 (ATC)
   Param_GBA16 : UDT 4;	//Sheet 12 (ATC)
   Param_GBA17 : UDT 4;	//Sheet 12 (ATC)
   Param_GBA18 : UDT 4;	//Sheet 12 (ATC)
   Param_GBA19 : UDT 4;	//Sheet 12 (ATC)
   Param_GBA20 : UDT 4;	//Sheet 12 (ATC)
   Param_GBA21 : UDT 4;	//Sheet 12 (ATC)
   Param_GBA22 : UDT 4;	//Sheet 12 (ATC)
   Param_GBA23 : UDT 4;	//Sheet 12 (ATC)
   Param_GBA24 : UDT 4;	//Sheet 12 (ATC)
   Param_GBA25 : UDT 4;	//Sheet 15 (ATC)
   Param_GBA26 : UDT 4;	//Sheet 15 (ATC)
   Param_GBA27 : UDT 4;	//Sheet 15 (ATC)
   Param_A136 : UDT 4;	//Sheet 17 (ATC)
   Param_127 : UDT 4;	//Sheet 17 (ATC)
   Param_GBA28 : UDT 4;	//Sheet 17 (ATC)
   Param_GBA29 : UDT 4;	//Sheet 17 (ATC)
   Param_GBA30 : UDT 4;	//Sheet 17 (ATC)
   Param_GBA31 : UDT 4;	//Sheet 17 (ATC)
   Param_686 : UDT 4;	//Sheet 25 (ATC)
   Param_685 : UDT 4;	//Sheet 25 (ATC)
   Param_325 : UDT 4;	//Sheet 29 (ATC)
   Param_326 : UDT 4;	//Sheet 29 (ATC)
   Param_327 : UDT 4;	//Sheet 29 (ATC)
   Param_328 : UDT 4;	//Sheet 29 (ATC)
   Param_329 : UDT 4;	//Sheet 29 (ATC)
   Param_399 : UDT 4;	//Sheet 29 (ATC)
   Param_377 : UDT 4;	//Sheet 31 (ATC)
   Param_378 : UDT 4;	//Sheet 31 (ATC)
   Param_GBA32 : UDT 4;	//Sheet 24 (ATC)
   Param_GBA33 : UDT 4;	//Sheet 24 (ATC)
   Param_GBA34 : UDT 4;	//Sheet 24 (ATC)
   Param_GBA35 : UDT 4;	//Sheet 24 (ATC)
   Param_GBA36 : UDT 4;	//Sheet 24 (ATC)
   Param_GBA37 : UDT 4;	//Sheet 24 (ATC)
   Param_GBA38 : UDT 4;	//Sheet 24 (ATC)
   Param_GBA39 : UDT 4;	//Sheet 24 (ATC)
   Param_GBA40 : UDT 4;	//Sheet 24 (ATC)
   Param_GBA41 : UDT 4;	//Sheet 24 (ATC)
   Param_381 : UDT 4;	//Sheet 33 (ATC)
   Param_311 : UDT 4;	//Sheet 35 (ATC)
   Param_A312 : UDT 4;	//Sheet 35 (ATC)
   Param_313 : UDT 4;	//Sheet 35 (ATC)
   Param_314 : UDT 4;	//Sheet 35 (ATC)
   Param_315 : UDT 4;	//Sheet 35 (ATC)
   Param_316 : UDT 4;	//Sheet 35 (ATC)
   Param_317 : UDT 4;	//Sheet 35 (ATC)
   Param_318 : UDT 4;	//Sheet 35 (ATC)
   Param_319 : UDT 4;	//Sheet 35 (ATC)
   Param_644 : UDT 4;	//Sheet 24 (ATC)
   Param_647 : UDT 4;	//Sheet 24 (ATC)
   Param_650 : UDT 4;	//Sheet 24 (ATC)
   Param_653 : UDT 4;	//Sheet 24 (ATC)
   Param_656 : UDT 4;	//Sheet 24 (ATC)
   Param_659 : UDT 4;	//Sheet 24 (ATC)
   Param_703 : UDT 4;	//Sheet 24 (ATC)
   Param_706 : UDT 4;	//Sheet 24 (ATC)
   Param_709 : UDT 4;	//Sheet 24 (ATC)
   Param_243 : UDT 4;	//Sheet 24 (ATC)
  END_STRUCT ;	
BEGIN
   Param_90.GAIN := 1.800000e+00;
   Param_90.BIAS := 3.200000e+01;
   Param_91.GAIN := 1.800000e+00;
   Param_91.BIAS := 3.200000e+01;
   Param_057.GAIN := 1.000000e+00;
   Param_92.GAIN := 3.937000e-01;
   Param_93.GAIN := 3.937000e-01;
   Param_88.GAIN := 1.800000e+00;
   Param_88.BIAS := 3.200000e+01;
   Param_055.GAIN := 1.800000e+00;
   Param_055.BIAS := 3.200000e+01;
   Param_790.GAIN := 1.527980e+00;
   Param_224.GAIN := -1.000000e+00;
   Param_224.BIAS := 1.500000e+03;
   Param_713.GAIN := 5.557000e-01;
   Param_711.GAIN := 5.557000e-01;
   Param_294.GAIN := 1.250000e-01;
   Param_295.GAIN := 2.875000e+00;
   Param_875.GAIN := 1.000000e+00;
   Param_143.GAIN := 5.555000e-01;
   Param_144.GAIN := -5.555000e-01;
   Param_466.GAIN := 1.800000e+00;
   Param_466.BIAS := 3.200000e+01;
   Param_468.GAIN := 1.800000e+00;
   Param_468.BIAS := 3.200000e+01;
   Param_A136.GAIN := 1.500000e-01;
   Param_127.GAIN := 1.000000e+00;
END_DATA_BLOCK

DATA_BLOCK "DELTAW-VALs"	// DB 6
AUTHOR : Sabeeh
VERSION : 0.1
  STRUCT
   Param_400 : UDT 5;	//Sheet 20 (RSM)
   Param_883 : UDT 5;	//Sheet 20 (RSM)
   Param_882 : UDT 5;	//Sheet 20 (RSM)
   Param_889 : UDT 5;	//Sheet 20 (RSM)
   Param_893 : UDT 5;	//Sheet 20 (RSM)
   Param_892 : UDT 5;	//Sheet 20 (RSM)
  END_STRUCT ;	
BEGIN
   Param_400.WT1 := 1.000000e+00;
   Param_400.WT2 := 1.000000e+00;
   Param_883.WT1 := 5.540000e-03;
   Param_883.WT2 := 5.540000e-03;
   Param_882.WT1 := 1.910000e-03;
   Param_882.WT2 := 1.910000e-03;
   Param_889.WT1 := 1.000000e+00;
   Param_889.WT2 := 1.000000e+00;
   Param_893.WT1 := 1.910000e-03;
   Param_893.WT2 := 1.910000e-03;
   Param_892.WT1 := 5.540000e-03;
   Param_892.WT2 := 5.540000e-03;
END_DATA_BLOCK

DATA_BLOCK "HILOLMTV-VALs"	// DB 7
AUTHOR : Sabeeh
VERSION : 0.1
  STRUCT
   Param_876 : UDT 6;	//Sheet 20 (RSM)
   Param_877 : UDT 6;	//Sheet 21 (RSM)
   Param_994 : UDT 6;	//Sheet 30 (ATC)
  END_STRUCT ;	
BEGIN
END_DATA_BLOCK

DATA_BLOCK "HILOMTR-VALs"	// DB 8
AUTHOR : Sabeeh
VERSION : 0.1
  STRUCT
   Param_X66D : UDT 7;	//Sheet 4 (RSM)
   Param_139 : UDT 7;	//Sheet 17 (ATC)
   Param_901 : UDT 7;	//Sheet 30 (ATC)
   Param_X60N : UDT 7;	//Sheet 35 (ATC)
  END_STRUCT ;	
BEGIN
   Param_X66D.HISP := 3.025000e+03;
   Param_X66D.HIDB := 5.000000e-01;
   Param_X66D.LOSP := 2.950000e+03;
   Param_X66D.LODB := 5.000000e-01;
   Param_139.HISP := 3.000000e+00;
   Param_139.HIDB := 5.000000e-01;
   Param_139.LOSP := -3.000000e+00;
   Param_139.LODB := 5.000000e-01;
END_DATA_BLOCK

DATA_BLOCK "AVALGEN"	// DB 9
AUTHOR : RJ
VERSION : 0.1
  STRUCT
   A392 : REAL  := 1.625000e+002;	//Sheet 2 (RSM)
   A200 : REAL ;	//Sheet 48 (ATC)
   A225 : REAL ;	//Sheet 48 (ATC)
   A601 : REAL ;	//Sheet 48 (ATC)
   A602 : REAL ;	//Sheet 48 (ATC)
   A603 : REAL ;	//Sheet 48 (ATC)
   A604 : REAL ;	//Sheet 48 (ATC)
   A56 : REAL ;	//Sheet 48 (ATC)
   A142 : REAL ;	//Sheet 48 (ATC)
   A143 : REAL ;	//Sheet 48 (ATC)
   A145 : REAL ;	//Sheet 48 (ATC)
   A147 : REAL ;	//Sheet 48 (ATC)
   A100 : REAL ;	//Sheet 48 (ATC)
   A150 : REAL ;	//Sheet 48 (ATC)
   A152 : REAL ;	//Sheet 48 (ATC)
   A153 : REAL ;	//Sheet 48 (ATC)
   A155 : REAL ;	//Sheet 48 (ATC)
   A157 : REAL ;	//Sheet 48 (ATC)
   A158 : REAL ;	//Sheet 48 (ATC)
   A160 : REAL ;	//Sheet 48 (ATC)
   A162 : REAL ;	//Sheet 48 (ATC)
   A163 : REAL ;	//Sheet 48 (ATC)
   A165 : REAL ;	//Sheet 48 (ATC)
   A167 : REAL ;	//Sheet 48 (ATC)
   A168 : REAL ;	//Sheet 48 (ATC)
   A170 : REAL ;	//Sheet 48 (ATC)
   A172 : REAL ;	//Sheet 48 (ATC)
   A173 : REAL ;	//Sheet 48 (ATC)
   A175 : REAL ;	//Sheet 48 (ATC)
   A177 : REAL ;	//Sheet 48 (ATC)
   A178 : REAL ;	//Sheet 48 (ATC)
   A180 : REAL ;	//Sheet 48 (ATC)
   A182 : REAL ;	//Sheet 48 (ATC)
   A183 : REAL ;	//Sheet 48 (ATC)
   A185 : REAL ;	//Sheet 48 (ATC)
   A995 : REAL ;	//Sheet 48 (ATC)
   A141 : REAL ;	//Sheet 48 (ATC)
   A140 : REAL ;	//Sheet 48 (ATC)
   A6 : REAL ;	//Sheet 49 (ATC)
   A7 : REAL ;	//Sheet 49 (ATC)
   A81 : REAL ;	//Sheet 49 (ATC)
   A82 : REAL ;	//Sheet 49 (ATC)
   A85 : REAL ;	//Sheet 49 (ATC)
   A86 : REAL ;	//Sheet 49 (ATC)
   A93 : REAL ;	//Sheet 49 (ATC)
   A94 : REAL ;	//Sheet 49 (ATC)
   A99 : REAL ;	//Sheet 49 (ATC)
   A101 : REAL ;	//Sheet 49 (ATC)
   A499 : REAL ;	//Sheet 49 (ATC)
   A110 : REAL ;	//Sheet 49 (ATC)
   A111 : REAL ;	//Sheet 49 (ATC)
   A118 : REAL ;	//Sheet 49 (ATC)
   A121 : REAL ;	//Sheet 49 (ATC)
   A148 : REAL ;	//Sheet 49 (ATC)
   A259 : REAL ;	//Sheet 49 (ATC)
   A308 : REAL ;	//Sheet 49 (ATC)
   A309 : REAL ;	//Sheet 49 (ATC)
   A310 : REAL ;	//Sheet 49 (ATC)
   A311 : REAL ;	//Sheet 49 (ATC)
   A359 : REAL ;	//Sheet 49 (ATC)
   A368 : REAL ;	//Sheet 49 (ATC)
   A373 : REAL ;	//Sheet 49 (ATC)
   A375 : REAL ;	//Sheet 49 (ATC)
   A376 : REAL ;	//Sheet 49 (ATC)
  END_STRUCT ;	
BEGIN
   A392 := 1.625000e+02;
END_DATA_BLOCK

DATA_BLOCK "DVALGEN"	// DB 10
AUTHOR : RJ
VERSION : 0.1
  STRUCT
   D22 : BOOL ;	//Sheet 2 (RSM). TRUE only if HP rotor T-ROOT grooves apply
   Q_Const : BOOL ;	//Constant quality used in QC blocks
   DTRUE : BOOL  := TRUE;	//Constant for TRUE value of BOOL
   DFALSE : BOOL ;	//Constant for FALSE value of BOOL
  END_STRUCT ;	
BEGIN
   DTRUE := TRUE;
END_DATA_BLOCK

DATA_BLOCK "RUNAVG_VALs_369_370"	// DB 11
AUTHOR : RJ
FAMILY : RSM
VERSION : 0.1
"RUNAVG"
BEGIN
END_DATA_BLOCK

DATA_BLOCK "HISIGMTV-VALs"	// DB 12
AUTHOR : Sabeeh
VERSION : 0.1
  STRUCT
   Param_121 : UDT 8;	//Sheet 4 (RSM)
   Param_228 : UDT 8;	//Sheet 8 (RSM)
   Param_393 : UDT 8;	//Sheet 19 (RSM)
   Param_398 : UDT 8;	//Sheet 19 (RSM)
   Param_008 : UDT 8;	//Sheet 12 (ATC)
   Param_043 : UDT 8;	//Sheet 12 (ATC)
   Param_009 : UDT 8;	//Sheet 12 (ATC)
   Param_045 : UDT 8;	//Sheet 12 (ATC)
   Param_012 : UDT 8;	//Sheet 12 (ATC)
   Param_046 : UDT 8;	//Sheet 12 (ATC)
   Param_015 : UDT 8;	//Sheet 12 (ATC)
   Param_047 : UDT 8;	//Sheet 12 (ATC)
   Param_016 : UDT 8;	//Sheet 12 (ATC)
   Param_048 : UDT 8;	//Sheet 12 (ATC)
   Param_018 : UDT 8;	//Sheet 12 (ATC)
   Param_049 : UDT 8;	//Sheet 12 (ATC)
   Param_112 : UDT 8;	//Sheet 12 (ATC)
   Param_113 : UDT 8;	//Sheet 12 (ATC)
   Param_052 : UDT 8;	//Sheet 12 (ATC)
   Param_031 : UDT 8;	//Sheet 12 (ATC)
   Param_032 : UDT 8;	//Sheet 12 (ATC)
   Param_075 : UDT 8;	//Sheet 12 (ATC)
   Param_038 : UDT 8;	//Sheet 12 (ATC)
   Param_076 : UDT 8;	//Sheet 12 (ATC)
   Param_241 : UDT 8;	//Sheet 12 (ATC)
   Param_077 : UDT 8;	//Sheet 12 (ATC)
   Param_041 : UDT 8;	//Sheet 12 (ATC)
   Param_078 : UDT 8;	//Sheet 12 (ATC)
   Param_042 : UDT 8;	//Sheet 12 (ATC)
   Param_079 : UDT 8;	//Sheet 12 (ATC)
   Param_AA : UDT 8;	//Sheet 12 (ATC)
   Param_CC : UDT 8;	//Sheet 12 (ATC)
   Param_114 : UDT 8;	//Sheet 12 (ATC)
   Param_115 : UDT 8;	//Sheet 12 (ATC)
   Param_116 : UDT 8;	//Sheet 12 (ATC)
   Param_117 : UDT 8;	//Sheet 12 (ATC)
   Param_360 : UDT 8;	//Sheet 12 (ATC)
   Param_361 : UDT 8;	//Sheet 12 (ATC)
   Param_XX : UDT 8;	//Sheet 12 (ATC)
   Param_YY : UDT 8;	//Sheet 12 (ATC)
   Param_362 : UDT 8;	//Sheet 12 (ATC)
   Param_363 : UDT 8;	//Sheet 12 (ATC)
   Param_364 : UDT 8;	//Sheet 12 (ATC)
   Param_365 : UDT 8;	//Sheet 12 (ATC)
   Param_366 : UDT 8;	//Sheet 12 (ATC)
   Param_367 : UDT 8;	//Sheet 12 (ATC)
   Param_369 : UDT 8;	//Sheet 12 (ATC)
   Param_370 : UDT 8;	//Sheet 12 (ATC)
   Param_371 : UDT 8;	//Sheet 12 (ATC)
   Param_372 : UDT 8;	//Sheet 12 (ATC)
   Param_UU : UDT 8;	//Sheet 12 (ATC)
   Param_VV2 : UDT 8;	//Sheet 12 (ATC)
   Param_098 : UDT 8;	//Sheet 15 (ATC)
   Param_273 : UDT 8;	//Sheet 15 (ATC)
   Param_097 : UDT 8;	//Sheet 15 (ATC)
   Param_272 : UDT 8;	//Sheet 15 (ATC)
   Param_102 : UDT 8;	//Sheet 15 (ATC)
   Param_103 : UDT 8;	//Sheet 15 (ATC)
   Param_137 : UDT 8;	//Sheet 17 (ATC)
   Param_415 : UDT 8;	//Sheet 25 (ATC)
   Param_862 : UDT 8;	//Sheet 25 (ATC)
   Param_331 : UDT 8;	//Sheet 25 (ATC)
   Param_343 : UDT 8;	//Sheet 25 (ATC)
   Param_864 : UDT 8;	//Sheet 25 (ATC)
   Param_281 : UDT 8;	//Sheet 25 (ATC)
   Param_332 : UDT 8;	//Sheet 25 (ATC)
   Param_344 : UDT 8;	//Sheet 25 (ATC)
   Param_867 : UDT 8;	//Sheet 25 (ATC)
   Param_282 : UDT 8;	//Sheet 25 (ATC)
   Param_333 : UDT 8;	//Sheet 25 (ATC)
   Param_345 : UDT 8;	//Sheet 25 (ATC)
   Param_870 : UDT 8;	//Sheet 25 (ATC)
   Param_283 : UDT 8;	//Sheet 25 (ATC)
   Param_334 : UDT 8;	//Sheet 25 (ATC)
   Param_346 : UDT 8;	//Sheet 25 (ATC)
   Param_873 : UDT 8;	//Sheet 25 (ATC)
   Param_284 : UDT 8;	//Sheet 25 (ATC)
   Param_335 : UDT 8;	//Sheet 25 (ATC)
   Param_347 : UDT 8;	//Sheet 25 (ATC)
   Param_379 : UDT 8;	//Sheet 31 (ATC)
   Param_383 : UDT 8;	//Sheet 31 (ATC)
   Param_A119 : UDT 8;	//Sheet 31 (ATC)
   Param_621 : UDT 8;	//Sheet 24 (ATC)
   Param_622 : UDT 8;	//Sheet 24 (ATC)
   Param_623 : UDT 8;	//Sheet 24 (ATC)
   Param_624 : UDT 8;	//Sheet 24 (ATC)
   Param_625 : UDT 8;	//Sheet 24 (ATC)
   Param_626 : UDT 8;	//Sheet 24 (ATC)
   Param_627 : UDT 8;	//Sheet 24 (ATC)
   Param_628 : UDT 8;	//Sheet 24 (ATC)
   Param_629 : UDT 8;	//Sheet 24 (ATC)
   Param_630 : UDT 8;	//Sheet 24 (ATC)
   Param_631 : UDT 8;	//Sheet 24 (ATC)
   Param_632 : UDT 8;	//Sheet 24 (ATC)
   Param_637 : UDT 8;	//Sheet 24 (ATC)
   Param_638 : UDT 8;	//Sheet 24 (ATC)
   Param_639 : UDT 8;	//Sheet 24 (ATC)
   Param_640 : UDT 8;	//Sheet 24 (ATC)
   Param_641 : UDT 8;	//Sheet 24 (ATC)
   Param_642 : UDT 8;	//Sheet 24 (ATC)
   Param_232 : UDT 8;	//Sheet 24 (ATC)
   Param_237 : UDT 8;	//Sheet 24 (ATC)
   Param_788 : UDT 8;	//Sheet 24 (ATC)
   Param_789 : UDT 8;	//Sheet 24 (ATC)
   Param_790 : UDT 8;	//Sheet 24 (ATC)
   Param_791 : UDT 8;	//Sheet 24 (ATC)
   Param_792 : UDT 8;	//Sheet 24 (ATC)
   Param_793 : UDT 8;	//Sheet 24 (ATC)
   Param_794 : UDT 8;	//Sheet 24 (ATC)
   Param_795 : UDT 8;	//Sheet 24 (ATC)
   Param_805 : UDT 8;	//Sheet 24 (ATC)
   Param_246 : UDT 8;	//Sheet 24 (ATC)
  END_STRUCT ;	
BEGIN
   Param_008.DBAN := 5.000000e+00;
   Param_043.DBAN := 5.000000e+00;
   Param_009.DBAN := 5.000000e+00;
   Param_045.DBAN := 5.000000e+00;
   Param_012.DBAN := 5.000000e+00;
   Param_046.DBAN := 5.000000e+00;
   Param_015.DBAN := 5.000000e+00;
   Param_047.DBAN := 5.000000e+00;
   Param_016.DBAN := 5.000000e+00;
   Param_048.DBAN := 5.000000e+00;
   Param_018.DBAN := 5.000000e+00;
   Param_049.DBAN := 5.000000e+00;
   Param_112.DBAN := 5.000000e+00;
   Param_113.DBAN := 5.000000e+00;
   Param_052.DBAN := 5.000000e+00;
   Param_031.DBAN := 5.000000e+00;
   Param_032.DBAN := 5.000000e+00;
   Param_075.DBAN := 5.000000e+00;
   Param_038.DBAN := 5.000000e+00;
   Param_076.DBAN := 5.000000e+00;
   Param_241.DBAN := 5.000000e+00;
   Param_077.DBAN := 5.000000e+00;
   Param_041.DBAN := 5.000000e+00;
   Param_078.DBAN := 5.000000e+00;
   Param_042.DBAN := 5.000000e+00;
   Param_079.DBAN := 5.000000e+00;
   Param_AA.DBAN := 5.000000e+00;
   Param_CC.DBAN := 5.000000e+00;
   Param_114.DBAN := 5.000000e+00;
   Param_115.DBAN := 5.000000e+00;
   Param_116.DBAN := 5.000000e+00;
   Param_117.DBAN := 5.000000e+00;
   Param_360.DBAN := 5.000000e+00;
   Param_361.DBAN := 5.000000e+00;
   Param_XX.DBAN := 5.000000e+00;
   Param_YY.DBAN := 5.000000e+00;
   Param_362.DBAN := 5.000000e+00;
   Param_363.DBAN := 5.000000e+00;
   Param_364.DBAN := 5.000000e+00;
   Param_365.DBAN := 5.000000e+00;
   Param_366.DBAN := 5.000000e+00;
   Param_367.DBAN := 5.000000e+00;
   Param_369.DBAN := 5.000000e+00;
   Param_370.DBAN := 5.000000e+00;
   Param_371.DBAN := 5.000000e+00;
   Param_372.DBAN := 5.000000e+00;
   Param_UU.DBAN := 5.000000e+00;
   Param_VV2.DBAN := 5.000000e+00;
   Param_137.DBAN := 5.000000e-01;
END_DATA_BLOCK

DATA_BLOCK "LOSIGMTV-VALs"	// DB 13
AUTHOR : Sabeeh
VERSION : 0.1
  STRUCT
   Param_395 : UDT 9;	//Sheet 19 (RSM)
   Param_095 : UDT 9;	//Sheet 15 (ATC)
   Param_270 : UDT 9;	//Sheet 15 (ATC)
   Param_096 : UDT 9;	//Sheet 15 (ATC)
   Param_271 : UDT 9;	//Sheet 15 (ATC)
   Param_106 : UDT 9;	//Sheet 15 (ATC)
   Param_108 : UDT 9;	//Sheet 15 (ATC)
   Param_089 : UDT 9;	//Sheet 15 (ATC)
   Param_090 : UDT 9;	//Sheet 15 (ATC)
   Param_993 : UDT 9;	//Sheet 25 (ATC)
   Param_863 : UDT 9;	//Sheet 25 (ATC)
   Param_337 : UDT 9;	//Sheet 25 (ATC)
   Param_350 : UDT 9;	//Sheet 25 (ATC)
   Param_865 : UDT 9;	//Sheet 25 (ATC)
   Param_866 : UDT 9;	//Sheet 25 (ATC)
   Param_338 : UDT 9;	//Sheet 25 (ATC)
   Param_351 : UDT 9;	//Sheet 25 (ATC)
   Param_868 : UDT 9;	//Sheet 25 (ATC)
   Param_869 : UDT 9;	//Sheet 25 (ATC)
   Param_339 : UDT 9;	//Sheet 25 (ATC)
   Param_352 : UDT 9;	//Sheet 25 (ATC)
   Param_A871 : UDT 9;	//Sheet 25 (ATC)
   Param_872 : UDT 9;	//Sheet 25 (ATC)
   Param_340 : UDT 9;	//Sheet 25 (ATC)
   Param_353 : UDT 9;	//Sheet 25 (ATC)
   Param_874 : UDT 9;	//Sheet 25 (ATC)
   Param_875 : UDT 9;	//Sheet 25 (ATC)
   Param_341 : UDT 9;	//Sheet 25 (ATC)
   Param_349 : UDT 9;	//Sheet 25 (ATC)
  END_STRUCT ;	
BEGIN
END_DATA_BLOCK

DATA_BLOCK "XLIMIT_VALs"	// DB 14
AUTHOR : Sabeeh
VERSION : 0.1
  STRUCT
   Param_X736 : UDT 10;	//Sheet 21 (RSM)
   Param_X301 : UDT 10;	//Sheet 7 (ATC)
   Param_X658 : UDT 10;	//Sheet 46 (ATC)
   Param_XA638 : UDT 10;	//Sheet 46 (ATC)
  END_STRUCT ;	
BEGIN
   Param_X736.GAIN := 1.000000e+00;
   Param_X736.SCLTOP := 1.000000e+04;
   Param_X736.SCLBTM := -1.000000e+04;
   Param_X301.GAIN := 1.800000e+00;
   Param_X301.BIAS := 3.200000e+01;
   Param_X301.SCLTOP := 1.000000e+03;
   Param_X658.GAIN := 1.000000e+00;
   Param_X658.SCLTOP := 1.000000e+02;
   Param_X658.SCLBTM := -1.000000e+02;
   Param_XA638.GAIN := 1.000000e+00;
   Param_XA638.SCLTOP := 1.000000e+02;
   Param_XA638.SCLBTM := -1.000000e+02;
END_DATA_BLOCK

DATA_BLOCK "AIFCTGEN_Vals"	// DB 15
AUTHOR : RJ
VERSION : 0.1
  STRUCT
   Param_880 : UDT 21;	//Sheet 17 (ATC)
   Param_881 : UDT 21;	//Sheet 17 (ATC)
   Param_600 : UDT 21;	//Sheet 20 (ATC)
   Param_455 : UDT 21;	//Sheet 46 (ATC)
   Param_456 : UDT 21;	//Sheet 46 (ATC)
  END_STRUCT ;	
BEGIN
   Param_880.R[2] := 2.499000e+03;
   Param_880.R[3] := 2.499500e+03;
   Param_880.R[4] := 3.450000e+03;
   Param_880.S[1] := 1.000000e+02;
   Param_880.S[2] := 1.000000e+02;
   Param_880.S[3] := 8.890000e+01;
   Param_880.S[4] := 5.500000e+00;
   Param_880.NMBP := 4;
   Param_881.R[2] := 3.250000e+01;
   Param_881.R[3] := 3.300000e+01;
   Param_881.R[4] := 3.250000e+02;
   Param_881.S[1] := 5.500000e+00;
   Param_881.S[2] := 5.500000e+00;
   Param_881.S[3] := 5.500000e+00;
   Param_881.S[4] := 5.500000e+00;
   Param_881.NMBP := 4;
   Param_600.R[1] := 1.000000e+03;
   Param_600.R[2] := 1.350000e+03;
   Param_600.S[1] := 2.032000e+02;
   Param_600.S[2] := 1.270000e+02;
   Param_600.NMBP := 2;
   Param_455.R[1] := 1.000000e+00;
   Param_455.R[2] := 2.000000e+00;
   Param_455.R[3] := 3.000000e+00;
   Param_455.R[4] := 4.000000e+00;
   Param_455.R[5] := 5.000000e+00;
   Param_455.R[6] := 6.000000e+00;
   Param_455.R[7] := 7.000000e+00;
   Param_455.R[8] := 8.000000e+00;
   Param_455.R[9] := 9.000000e+00;
   Param_455.S[1] := 1.000000e+00;
   Param_455.S[2] := 2.000000e+00;
   Param_455.S[3] := 3.000000e+00;
   Param_455.S[4] := 4.000000e+00;
   Param_455.S[5] := 5.000000e+00;
   Param_455.S[6] := 6.000000e+00;
   Param_455.S[7] := 7.000000e+00;
   Param_455.S[8] := 8.000000e+00;
   Param_455.S[9] := 9.000000e+00;
   Param_455.NMBP := 5;
   Param_456.R[1] := 1.000000e+00;
   Param_456.R[2] := 2.000000e+00;
   Param_456.R[3] := 3.000000e+00;
   Param_456.R[4] := 4.000000e+00;
   Param_456.R[5] := 5.000000e+00;
   Param_456.R[6] := 6.000000e+00;
   Param_456.R[7] := 7.000000e+00;
   Param_456.R[8] := 8.000000e+00;
   Param_456.R[9] := 9.000000e+00;
   Param_456.S[1] := 1.000000e+00;
   Param_456.S[2] := 2.000000e+00;
   Param_456.S[3] := 3.000000e+00;
   Param_456.S[4] := 4.000000e+00;
   Param_456.S[5] := 5.000000e+00;
   Param_456.S[6] := 6.000000e+00;
   Param_456.S[7] := 7.000000e+00;
   Param_456.S[8] := 8.000000e+00;
   Param_456.S[9] := 9.000000e+00;
   Param_456.NMBP := 5;
END_DATA_BLOCK

DATA_BLOCK "MULTGB_VALs"	// DB 16
AUTHOR : Sabeeh
VERSION : 0.1
  STRUCT
   Param_794 : UDT 11;	//Sheet 3 (RSM)
   Param_211 : UDT 11;	//Sheet 3 (RSM)
   Param_212 : UDT 11;	//Sheet 3 (RSM)
   Param_105 : UDT 11;	//Sheet 4 (RSM)
   Param_104 : UDT 11;	//Sheet 4 (RSM)
   Param_103 : UDT 11;	//Sheet 4 (RSM)
   Param_310 : UDT 11;	//Sheet 9 (RSM)
   Param_311 : UDT 11;	//Sheet 9 (RSM)
   Param_313 : UDT 11;	//Sheet 9 (RSM)
   Param_414 : UDT 11;	//Sheet 8 (RSM)
   Param_413 : UDT 11;	//Sheet 8 (RSM)
   Param_416 : UDT 11;	//Sheet 8 (RSM)
   Param_417 : UDT 11;	//Sheet 8 (RSM)
   Param_225 : UDT 11;	//Sheet 8 (RSM)
   Param_167 : UDT 11;	//Sheet 13 (RSM)
   Param_170 : UDT 11;	//Sheet 13 (RSM)
   Param_172 : UDT 11;	//Sheet 13 (RSM)
   Param_044 : UDT 11;	//Sheet 20 (RSM)
   Param_042 : UDT 11;	//Sheet 20 (RSM)
   Param_885 : UDT 11;	//Sheet 20 (RSM)
   Param_890 : UDT 11;	//Sheet 20 (RSM)
   Param_891 : UDT 11;	//Sheet 20 (RSM)
   Param_895 : UDT 11;	//Sheet 20 (RSM)
  END_STRUCT ;	
BEGIN
   Param_794.GAIN := 1.000000e+00;
   Param_211.GAIN := 1.000000e+00;
   Param_212.GAIN := 1.000000e+00;
   Param_105.GAIN := 1.000000e+00;
   Param_104.GAIN := 1.000000e+00;
   Param_103.GAIN := 1.000000e+00;
   Param_310.GAIN := 1.000000e+00;
   Param_311.GAIN := 1.000000e+00;
   Param_313.GAIN := 1.000000e+00;
   Param_414.GAIN := 1.000000e+00;
   Param_413.GAIN := 1.000000e+00;
   Param_416.GAIN := 1.000000e+00;
   Param_417.GAIN := 1.000000e+00;
   Param_225.GAIN := 1.000000e+00;
   Param_167.GAIN := 1.000000e+00;
   Param_170.GAIN := 1.000000e+00;
   Param_172.GAIN := 1.000000e+00;
   Param_044.GAIN := 1.000000e+00;
   Param_042.GAIN := 1.000000e+00;
   Param_885.GAIN := 1.000000e+00;
   Param_890.GAIN := 1.000000e+00;
   Param_891.GAIN := 1.000000e+00;
   Param_895.GAIN := 1.000000e+00;
END_DATA_BLOCK

DATA_BLOCK "SUM2W_VALs"	// DB 17
AUTHOR : Sabeeh
VERSION : 0.1
  STRUCT
   Param_371 : UDT 12;	//Sheet 3 (RSM)
   Param_372 : UDT 12;	//Sheet 3 (RSM)
   Param_792 : UDT 12;	//Sheet 3 (RSM)
   Param_312 : UDT 12;	//IN1 of Block 312 should have a -ve weight w.r.f sheet 9 (RSM).
   Param_160 : UDT 12;	//Sheet 9 (RSM)
   Param_410 : UDT 12;	//Sheet 8 (RSM)
   Param_411 : UDT 12;	//Sheet 8 (RSM)
   Param_412 : UDT 12;	//Sheet 8 (RSM)
   Param_415 : UDT 12;	//Sheet 8 (RSM)
   Param_226 : UDT 12;	//Sheet 8 (RSM)
   Param_161 : UDT 12;	//Sheet 11 (RSM)
   Param_168 : UDT 12;	//IN2 should have -ve weight as shown in sheet 13 (RSM).
   Param_169 : UDT 12;	//IN2 should have -ve weight as shown in sheet 13 (RSM).
   Param_173 : UDT 12;	//Sheet 13 (RSM)
   Param_174 : UDT 12;	//IN2 should have -ve weight as shown in sheet 13 (RSM).
   Param_171 : UDT 12;	//IN2 should have -ve weight as shown in sheet 13 (RSM).
   Param_293 : UDT 12;	//Sheet 16 (RSM)
   Param_296 : UDT 12;	//IN1 should have -ve weight as shown in sheet 16 (RSM).
   Param_884 : UDT 12;	//Sheet 20 (RSM)
   Param_894 : UDT 12;	//Sheet 20 (RSM)
   Param_323 : UDT 12;	//IN2 should have -ve weight as shown in sheet 21 (RSM).
   Param_A883 : UDT 12;	//Sheet 17 (ATC)
   Param_138 : UDT 12;	//IN2 should have -ve weight as shown in sheet 17 (ATC).
   Param_900 : UDT 12;	//Sheet 30 (ATC)
   Param_998 : UDT 12;	//Sheet 35 (ATC)
   Param_997 : UDT 12;	//Sheet 35 (ATC)
   Param_996 : UDT 12;	//Sheet 35 (ATC)
   Param_999 : UDT 12;	//Sheet 35 (ATC)
   Param_643 : UDT 12;	//Sheet 24 (ATC)
   Param_646 : UDT 12;	//Sheet 24 (ATC)
   Param_649 : UDT 12;	//Sheet 24 (ATC)
   Param_652 : UDT 12;	//Sheet 24 (ATC)
   Param_655 : UDT 12;	//Sheet 24 (ATC)
   Param_658 : UDT 12;	//Sheet 24 (ATC)
   Param_702 : UDT 12;	//Sheet 24 (ATC)
   Param_705 : UDT 12;	//Sheet 24 (ATC)
   Param_708 : UDT 12;	//Sheet 24 (ATC)
   Param_242 : UDT 12;	//Sheet 24 (ATC)
   Param_645 : UDT 12;	//Sheet 24 (ATC)
   Param_648 : UDT 12;	//Sheet 24 (ATC)
   Param_651 : UDT 12;	//Sheet 24 (ATC)
   Param_654 : UDT 12;	//Sheet 24 (ATC)
   Param_657 : UDT 12;	//Sheet 24 (ATC)
   Param_660 : UDT 12;	//Sheet 24 (ATC)
   Param_704 : UDT 12;	//Sheet 24 (ATC)
   Param_707 : UDT 12;	//Sheet 24 (ATC)
   Param_710 : UDT 12;	//Sheet 24 (ATC)
   Param_244 : UDT 12;	//Sheet 24 (ATC)
  END_STRUCT ;	
BEGIN
   Param_371.WT1 := 1.000000e+00;
   Param_371.WT2 := -1.000000e+00;
   Param_372.WT1 := 1.000000e+00;
   Param_372.WT2 := -1.000000e+00;
   Param_792.WT1 := 8.190000e+02;
   Param_792.WT2 := 4.910000e-01;
   Param_312.WT1 := -1.000000e+00;
   Param_312.WT2 := 1.000000e+00;
   Param_160.WT1 := 1.000000e+00;
   Param_160.WT2 := 1.000000e+00;
   Param_410.WT1 := 1.000000e+00;
   Param_410.WT2 := 1.000000e+00;
   Param_411.WT1 := 1.000000e+00;
   Param_411.WT2 := 1.000000e+00;
   Param_412.WT1 := 1.000000e+00;
   Param_412.WT2 := 1.000000e+00;
   Param_415.WT1 := 1.000000e+00;
   Param_415.WT2 := 1.000000e+00;
   Param_226.WT1 := 1.000000e+00;
   Param_226.WT2 := -1.000000e+00;
   Param_161.WT1 := 1.000000e+00;
   Param_161.WT2 := 1.000000e+00;
   Param_168.WT1 := 1.000000e+00;
   Param_168.WT2 := -1.000000e+00;
   Param_169.WT1 := 1.000000e+00;
   Param_169.WT2 := -1.000000e+00;
   Param_173.WT1 := 1.000000e+00;
   Param_173.WT2 := 1.000000e+00;
   Param_174.WT1 := 1.000000e+00;
   Param_174.WT2 := -1.000000e+00;
   Param_171.WT1 := 1.000000e+00;
   Param_171.WT2 := -1.000000e+00;
   Param_293.WT1 := 1.000000e+00;
   Param_293.WT2 := 1.000000e+00;
   Param_296.WT1 := -1.000000e+00;
   Param_296.WT2 := 1.000000e+00;
   Param_884.WT1 := 1.000000e+00;
   Param_884.WT2 := 1.000000e+00;
   Param_894.WT1 := 1.000000e+00;
   Param_894.WT2 := 1.000000e+00;
   Param_323.WT1 := 1.000000e+00;
   Param_323.WT2 := -1.000000e+00;
   Param_A883.WT1 := 1.000000e+00;
   Param_A883.WT2 := -1.000000e+00;
   Param_138.WT1 := 1.000000e+00;
   Param_138.WT2 := -1.000000e+00;
END_DATA_BLOCK

DATA_BLOCK "RATEMTR_VALs"	// DB 18
AUTHOR : Sabeeh
VERSION : 0.1
  STRUCT
   Param_599 : UDT 13;	//Sheet 21 (RSM)
   Param_600 : UDT 13;	//Sheet 21 (RSM)
  END_STRUCT ;	
BEGIN
   Param_599.PRATE := 1.000000e+03;
   Param_599.NRATE := 8.000000e-03;
   Param_600.PRATE := 8.000000e-03;
   Param_600.NRATE := 1.000000e+03;
END_DATA_BLOCK

DATA_BLOCK "XSUM_VALs"	// DB 19
AUTHOR : Sabeeh
VERSION : 0.1
  STRUCT
   Param_X111 : UDT 14;	//PV gain of the block should be -ve as shown in sheet 17 (RSM)
   Param_X731 : UDT 14;	//PV gain of the block should be -ve as shown in sheet 17 (RSM)
   Param_X113 : UDT 14;	//PV gain of the block should be -ve as shown in sheet 17 (RSM)
   Param_X115 : UDT 14;	//PV gain of the block should be -ve as shown in sheet 17 (RSM)
   Param_X112 : UDT 14;	//PV gain of the block should be -ve as shown in sheet 17 (RSM)
   Param_X114 : UDT 14;	//PV gain of the block should be -ve as shown in sheet 17 (RSM)
   Param_X116 : UDT 14;	//PV gain of the block should be -ve as shown in sheet 17 (RSM)
   Param_X091 : UDT 14;	//PV gain of the block should be -ve as shown in sheet 17 (RSM)
   Param_X121 : UDT 14;	//Sheet 18 (RSM)
   Param_X123 : UDT 14;	//Sheet 18 (RSM)
   Param_X132 : UDT 14;	//Sheet 18 (RSM)
   Param_X134 : UDT 14;	//Sheet 18 (RSM)
   Param_X141 : UDT 14;	//PV gain of the block should be -ve as shown in sheet 18 (RSM)
   Param_X124 : UDT 14;	//PV gain of the block should be -ve as shown in sheet 18 (RSM)
   Param_X142 : UDT 14;	//PV gain of the block should be -ve as shown in sheet 18 (RSM)
   Param_X144 : UDT 14;	//PV gain of the block should be -ve as shown in sheet 18 (RSM)
   Param_X732 : UDT 14;	//PV gain of the block should be -ve as shown in sheet 21 (RSM)
   Param_X431 : UDT 14;	//Sheet 15 (ATC)
   Param_X191 : UDT 14;	//Sheet 31 (ATC)
   Param_X601 : UDT 14;	//PV gain of the block should be -ve as shown in sheet 35 (ATC)
   Param_X602 : UDT 14;	//PV gain of the block should be -ve as shown in sheet 35 (ATC)
   Param_X656 : UDT 14;	//Sheet 46 (ATC)
   Param_X651 : UDT 14;	//PV gain of the block should be -ve as shown in sheet 46 (ATC)
  END_STRUCT ;	
BEGIN
   Param_X111.PVGAIN := -1.000000e+00;
   Param_X111.CASGAIN := 1.000000e+00;
   Param_X111.SCALETOP := 9.999900e+04;
   Param_X111.SCALEBOT := -9.999900e+04;
   Param_X731.PVGAIN := -7.500000e-01;
   Param_X731.CASGAIN := 1.000000e+00;
   Param_X731.SCALETOP := 9.999900e+04;
   Param_X731.SCALEBOT := -9.999900e+04;
   Param_X113.PVGAIN := -8.500000e-01;
   Param_X113.CASGAIN := 1.000000e+00;
   Param_X113.SCALETOP := 9.999900e+04;
   Param_X113.SCALEBOT := -9.999900e+04;
   Param_X115.PVGAIN := -9.000000e-01;
   Param_X115.CASGAIN := 1.000000e+00;
   Param_X115.SCALETOP := 9.999900e+04;
   Param_X115.SCALEBOT := -9.999900e+04;
   Param_X112.PVGAIN := -1.000000e+00;
   Param_X112.CASGAIN := 1.000000e+00;
   Param_X112.SCALETOP := 9.999900e+04;
   Param_X112.SCALEBOT := -9.999900e+04;
   Param_X114.PVGAIN := -7.500000e-01;
   Param_X114.CASGAIN := 1.000000e+00;
   Param_X114.SCALETOP := 9.999900e+04;
   Param_X114.SCALEBOT := -9.999900e+04;
   Param_X116.PVGAIN := -5.000000e-01;
   Param_X116.CASGAIN := 1.000000e+00;
   Param_X116.SCALETOP := 9.999900e+04;
   Param_X116.SCALEBOT := -9.999900e+04;
   Param_X091.PVGAIN := -1.000000e+00;
   Param_X091.CASGAIN := 1.000000e+00;
   Param_X091.SCALETOP := 9.999900e+04;
   Param_X091.SCALEBOT := -9.999900e+04;
   Param_X121.PVGAIN := 1.000000e+00;
   Param_X121.CASGAIN := -1.000000e+00;
   Param_X121.SCALETOP := 9.999900e+04;
   Param_X121.SCALEBOT := -9.999900e+04;
   Param_X123.PVGAIN := 1.000000e-05;
   Param_X123.CASGAIN := 1.000000e-05;
   Param_X123.SCALETOP := 9.999900e+04;
   Param_X123.SCALEBOT := -9.999900e+04;
   Param_X132.PVGAIN := 1.000000e+00;
   Param_X132.CASGAIN := 1.000000e+00;
   Param_X132.SCALETOP := 9.999900e+04;
   Param_X132.SCALEBOT := -9.999900e+04;
   Param_X134.PVGAIN := 1.000000e+00;
   Param_X134.CASGAIN := 1.000000e+00;
   Param_X134.SCALETOP := 9.999900e+04;
   Param_X134.SCALEBOT := -9.999900e+04;
   Param_X141.PVGAIN := -1.000000e+00;
   Param_X141.CASGAIN := 1.000000e+00;
   Param_X141.SCALETOP := 9.999900e+04;
   Param_X141.SCALEBOT := -9.999900e+04;
   Param_X124.PVGAIN := -1.000000e-05;
   Param_X124.CASGAIN := 1.000000e-06;
   Param_X124.SCALETOP := 9.999900e+04;
   Param_X124.SCALEBOT := -9.999900e+04;
   Param_X142.PVGAIN := -5.000000e-01;
   Param_X142.CASGAIN := 1.000000e+00;
   Param_X142.SCALETOP := 9.999900e+04;
   Param_X142.SCALEBOT := -9.999900e+04;
   Param_X144.PVGAIN := -7.500000e-01;
   Param_X144.CASGAIN := 1.000000e+00;
   Param_X144.SCALETOP := 9.999900e+04;
   Param_X144.SCALEBOT := -9.999900e+04;
   Param_X732.PVGAIN := -1.000000e+00;
   Param_X732.CASGAIN := 1.000000e+00;
   Param_X732.SCALETOP := 9.999900e+04;
   Param_X732.SCALEBOT := -9.999900e+04;
   Param_X431.PVGAIN := 2.667000e+00;
   Param_X431.CASGAIN := -1.667000e+00;
   Param_X431.SCALETOP := 9.999900e+04;
   Param_X431.SCALEBOT := -9.999900e+04;
END_DATA_BLOCK

DATA_BLOCK "XTRANSF_VALs"	// DB 20
AUTHOR : Sabeeh
VERSION : 0.1
  STRUCT
   Param_X151 : UDT 15;	//Sheet 18 (RSM)
   Param_X152 : UDT 15;	//Sheet 18 (RSM)
   Param_X742 : UDT 15;	//Sheet 21 (RSM)
   Param_X734 : UDT 15;	//Sheet 21 (RSM)
   Param_X712 : UDT 15;	//Sheet 24 (RSM)
   Param_X715 : UDT 15;	//Sheet 24 (RSM)
   Param_X717 : UDT 15;	//Sheet 24 (RSM)
   Param_X721 : UDT 15;	//Sheet 24 (RSM)
   Param_X723 : UDT 15;	//Sheet 24 (RSM)
   Param_X725 : UDT 15;	//Sheet 24 (RSM)
   Param_X741 : UDT 15;	//Sheet 24 (RSM)
   Param_X743 : UDT 15;	//Sheet 24 (RSM)
   Param_X701 : UDT 15;	//Sheet 24 (RSM)
   Param_X707 : UDT 15;	//Sheet 24 (RSM)
   Param_X171 : UDT 15;	//Sheet 24 (RSM)
   Param_X652 : UDT 15;	//Sheet 46 (ATC)
   Param_X654 : UDT 15;	//Sheet 46 (ATC)
   Param_X631 : UDT 15;	//Sheet 46 (ATC)
   Param_X633 : UDT 15;	//Sheet 46 (ATC)
   Param_X635 : UDT 15;	//Sheet 46 (ATC)
   Param_X637 : UDT 15;	//Sheet 46 (ATC)
   Param_X638 : UDT 15;	//Sheet 46 (ATC)
  END_STRUCT ;	
BEGIN
   Param_X151.PV_YGAIN := 1.000000e+00;
   Param_X151.CAS_NGAIN := 1.000000e+00;
   Param_X151.SCALETOP := 9.999900e+04;
   Param_X151.SCALEBOT := -9.999900e+04;
   Param_X152.PV_YGAIN := 1.000000e+00;
   Param_X152.CAS_NGAIN := 1.000000e+00;
   Param_X152.SCALETOP := 9.999900e+04;
   Param_X152.SCALEBOT := -9.999900e+04;
   Param_X742.PV_YGAIN := 1.000000e+00;
   Param_X742.CAS_NGAIN := 1.000000e+00;
   Param_X742.SCALETOP := 9.999900e+04;
   Param_X742.SCALEBOT := -9.999900e+04;
   Param_X734.PV_YGAIN := 1.000000e+00;
   Param_X734.CAS_NGAIN := 1.000000e+00;
   Param_X734.SCALETOP := 9.999900e+04;
   Param_X734.SCALEBOT := -9.999900e+04;
   Param_X712.PV_YGAIN := 1.000000e+00;
   Param_X712.CAS_NGAIN := 1.000000e+00;
   Param_X712.SCALETOP := 9.999900e+04;
   Param_X712.SCALEBOT := -9.999900e+04;
   Param_X715.PV_YGAIN := 1.000000e+00;
   Param_X715.CAS_NGAIN := 1.000000e+00;
   Param_X715.SCALETOP := 9.999900e+04;
   Param_X715.SCALEBOT := -9.999900e+04;
   Param_X717.PV_YGAIN := 1.000000e+00;
   Param_X717.CAS_NGAIN := 1.000000e+00;
   Param_X717.SCALETOP := 9.999900e+04;
   Param_X717.SCALEBOT := -9.999900e+04;
   Param_X721.PV_YGAIN := 1.000000e+00;
   Param_X721.CAS_NGAIN := 1.000000e+00;
   Param_X721.SCALETOP := 9.999900e+04;
   Param_X721.SCALEBOT := -9.999900e+04;
   Param_X723.PV_YGAIN := 1.000000e+00;
   Param_X723.CAS_NGAIN := 1.000000e+00;
   Param_X723.SCALETOP := 9.999900e+04;
   Param_X723.SCALEBOT := -9.999900e+04;
   Param_X725.PV_YGAIN := 1.000000e+00;
   Param_X725.CAS_NGAIN := 1.000000e+00;
   Param_X725.SCALETOP := 1.000000e+08;
   Param_X725.SCALEBOT := -1.000000e+07;
   Param_X741.PV_YGAIN := 1.000000e-05;
   Param_X741.PV_YBIAS := 2.250000e+03;
   Param_X741.CAS_NGAIN := 1.000000e+00;
   Param_X741.SCALETOP := 9.999000e+03;
   Param_X741.SCALEBOT := -1.000000e+02;
   Param_X743.PV_YGAIN := 1.000000e+00;
   Param_X743.CAS_NGAIN := 1.000000e+00;
   Param_X743.SCALETOP := 9.999000e+03;
   Param_X743.SCALEBOT := -1.000000e+02;
   Param_X701.PV_YGAIN := 1.000000e+00;
   Param_X701.PV_YBIAS := 3.000000e+03;
   Param_X701.CAS_NGAIN := 1.000000e+00;
   Param_X701.SCALETOP := 9.999900e+04;
   Param_X701.SCALEBOT := -9.999900e+04;
   Param_X707.PV_YGAIN := 1.000000e+00;
   Param_X707.PV_YBIAS := 5.200000e+02;
   Param_X707.CAS_NGAIN := 1.000000e+00;
   Param_X707.SCALETOP := 9.999900e+04;
   Param_X707.SCALEBOT := -9.999900e+04;
   Param_X171.PV_YGAIN := 1.000000e+00;
   Param_X171.CAS_NGAIN := 1.000000e+00;
   Param_X171.SCALETOP := 9.999900e+04;
   Param_X171.SCALEBOT := -9.999900e+04;
END_DATA_BLOCK

DATA_BLOCK "XHISEL_VALs"	// DB 21
AUTHOR : RJ
VERSION : 0.1
  STRUCT
   Param_X081 : UDT 16;	//Sheet 4 (RSM)
  END_STRUCT ;	
BEGIN
   Param_X081.PV_GAIN := 1.000000e+00;
   Param_X081.CAS_GAIN := 1.000000e+00;
   Param_X081.SCALE_TOP := 1.000000e+03;
   Param_X081.SCALE_BOT := -1.000000e+02;
END_DATA_BLOCK

DATA_BLOCK "AIN_VALs_TEMP_100"	// DB 22
AUTHOR : RJ
VERSION : 0.1
"AIN"
BEGIN
END_DATA_BLOCK

DATA_BLOCK "DIVIDEGB_VALs"	// DB 23
AUTHOR : RJ
VERSION : 0.1
  STRUCT
   Param_793 : UDT 22;	//Sheet 3 (RSM)
   Param_227 : UDT 22;	//Sheet 8 (RSM)
   Param_165 : UDT 22;	//Sheet 12 (RSM)
  END_STRUCT ;	
BEGIN
   Param_793.GAIN := 1.000000e+00;
   Param_227.GAIN := 1.000000e+00;
   Param_165.GAIN := 1.000000e+00;
END_DATA_BLOCK

DATA_BLOCK "AIN_VALs_TEMP_286"	// DB 24
AUTHOR : RJ
VERSION : 0.1
"AIN"
BEGIN
END_DATA_BLOCK

DATA_BLOCK "POLY_VALs"	// DB 25
AUTHOR : RJ
VERSION : 0.1
  STRUCT
   Param_217 : UDT 23;	//Sheet 3 (RSM)
   Param_858 : UDT 23;	//Sheet 4 (RSM)
  END_STRUCT ;	
BEGIN
   Param_217.CX0 := 1.340000e+02;
   Param_217.CX1 := 8.699170e+00;
   Param_217.CX2 := -2.837170e-01;
   Param_217.CX3 := 5.304000e-03;
   Param_217.CX4 := -3.900000e-05;
   Param_858.CX0 := 2.997210e+02;
   Param_858.CX1 := -1.001740e-01;
   Param_858.CX2 := 1.760000e-04;
END_DATA_BLOCK

DATA_BLOCK "SUM4W_VALs"	// DB 26
AUTHOR : Sabeeh
VERSION : 0.1
  STRUCT
   Param_857 : UDT 20;	//Sheet 3 (RSM)
   Param_314 : UDT 20;	//Sheet 9 (RSM)
   Param_326 : UDT 20;	//Sheet 9 (RSM)
   Param_329 : UDT 20;	//Sheet 9 (RSM)
   Param_332 : UDT 20;	//Sheet 9 (RSM)
   Param_335 : UDT 20;	//Sheet 9 (RSM)
   Param_338 : UDT 20;	//Sheet 10 (RSM)
   Param_341 : UDT 20;	//Sheet 10 (RSM)
   Param_344 : UDT 20;	//Sheet 10 (RSM)
   Param_347 : UDT 20;	//Sheet 10 (RSM)
   Param_350 : UDT 20;	//Sheet 10 (RSM)
   Param_353 : UDT 20;	//Sheet 10 (RSM)
   Param_356 : UDT 20;	//Sheet 10 (RSM)
   Param_359 : UDT 20;	//Sheet 10 (RSM)
   Param_362 : UDT 20;	//Sheet 10 (RSM)
   Param_376 : UDT 20;	//Sheet 10 (RSM)
   Param_301 : UDT 20;	//Sheet 11 (RSM)
   Param_304 : UDT 20;	//Sheet 11 (RSM)
   Param_407 : UDT 20;	//Sheet 15 (ATC)
   Param_408 : UDT 20;	//Sheet 15 (ATC)
   Param_A413 : UDT 20;	//Sheet 15 (ATC)
   Param_A414 : UDT 20;	//Sheet 15 (ATC)
  END_STRUCT ;	
BEGIN
   Param_857.WT1 := 1.000000e+00;
   Param_857.WT2 := -4.788660e+01;
   Param_857.WT3 := 6.274270e+00;
   Param_857.WT4 := 1.000000e+00;
   Param_314.WT1 := 1.000000e+00;
   Param_314.WT2 := 1.000000e+00;
   Param_314.WT3 := 1.383240e-02;
   Param_326.WT1 := 7.203350e-02;
   Param_326.WT2 := 8.598130e-01;
   Param_326.WT3 := 6.815350e-02;
   Param_329.WT1 := 7.214720e-02;
   Param_329.WT2 := 8.598130e-01;
   Param_329.WT3 := 6.809800e-02;
   Param_332.WT1 := 7.227510e-02;
   Param_332.WT2 := 8.598130e-01;
   Param_332.WT3 := 6.791190e-02;
   Param_335.WT1 := 7.241990e-02;
   Param_335.WT2 := 8.598130e-01;
   Param_335.WT3 := 6.776710e-02;
   Param_338.WT1 := 7.258530e-02;
   Param_338.WT2 := 8.598130e-01;
   Param_338.WT3 := 6.760170e-02;
   Param_341.WT1 := 7.277600e-02;
   Param_341.WT2 := 8.598130e-01;
   Param_341.WT3 := 6.741100e-02;
   Param_344.WT1 := 7.299840e-02;
   Param_344.WT2 := 8.598130e-01;
   Param_344.WT3 := 6.718870e-02;
   Param_347.WT1 := 7.326090e-02;
   Param_347.WT2 := 8.598130e-01;
   Param_347.WT3 := 6.692610e-02;
   Param_350.WT1 := 3.575600e-02;
   Param_350.WT2 := 8.598130e-01;
   Param_350.WT3 := 6.661140e-02;
   Param_353.WT1 := 7.395970e-02;
   Param_353.WT2 := 8.598130e-01;
   Param_353.WT3 := 6.622730e-02;
   Param_356.WT1 := 7.443910e-02;
   Param_356.WT2 := 8.598130e-01;
   Param_356.WT3 := 6.574790e-02;
   Param_359.WT1 := 7.505420e-02;
   Param_359.WT2 := 8.598130e-01;
   Param_359.WT3 := 6.513280e-02;
   Param_362.WT1 := 7.587210e-02;
   Param_362.WT2 := 8.598130e-01;
   Param_362.WT3 := 6.431490e-02;
   Param_376.WT1 := 7.701300e-02;
   Param_376.WT2 := 8.598130e-01;
   Param_376.WT3 := 6.317400e-02;
   Param_301.WT1 := 7.871520e-02;
   Param_301.WT2 := 8.598130e-01;
   Param_301.WT3 := 6.147180e-02;
   Param_304.WT1 := 1.507590e-02;
   Param_304.WT2 := 8.492410e-01;
   Param_407.WT1 := 1.000000e+00;
   Param_407.WT2 := 1.000000e+00;
   Param_408.WT1 := 1.000000e+00;
   Param_408.WT2 := 1.000000e+00;
   Param_A413.WT1 := 1.000000e+00;
   Param_A413.WT2 := 1.000000e+00;
   Param_A414.WT1 := 1.000000e+00;
   Param_A414.WT2 := 1.000000e+00;
END_DATA_BLOCK

DATA_BLOCK "SUM8W_VALs"	// DB 27
AUTHOR : RJ
VERSION : 0.1
  STRUCT
   Param_791 : UDT 24;	//Sheet 3 (RSM)
   Param_106 : UDT 24;	//Sheet 4 (RSM)
   Param_162 : UDT 24;	//Sheet 12 (RSM)
   Param_163 : UDT 24;	//Sheet 12 (RSM)
   Param_164 : UDT 24;	//Sheet 12 (RSM)
   Param_291 : UDT 24;	//Sheet 16 (RSM)
   Param_292 : UDT 24;	//Sheet 16 (RSM)
  END_STRUCT ;	
BEGIN
   Param_791.WT1 := 2.040100e-06;
   Param_791.WT2 := 2.706060e-09;
   Param_791.WT3 := 1.661860e-09;
   Param_791.WT4 := -2.017570e-13;
   Param_791.WT6 := 1.000000e+00;
   Param_791.WT7 := 1.000000e+00;
   Param_791.WT8 := 1.000000e+00;
   Param_106.WT1 := 3.368460e-02;
   Param_106.WT2 := 9.695520e-03;
   Param_106.WT3 := -2.586220e-06;
   Param_106.WT4 := 2.256890e+00;
   Param_106.WT5 := 5.360000e+02;
   Param_106.WT6 := 1.500000e+03;
   Param_162.WT1 := 3.807910e-01;
   Param_162.WT2 := 3.712240e-01;
   Param_162.WT3 := 6.907460e-01;
   Param_162.WT4 := 6.502690e-01;
   Param_162.WT5 := 6.097910e-01;
   Param_162.WT6 := 5.693140e-01;
   Param_162.WT7 := 5.288360e-01;
   Param_162.WT8 := 4.883590e-01;
   Param_163.WT1 := 4.478810e-01;
   Param_163.WT2 := 4.074040e-01;
   Param_163.WT3 := 3.669260e-01;
   Param_163.WT4 := 3.264490e-01;
   Param_163.WT5 := 2.859710e-01;
   Param_163.WT6 := 2.454940e-01;
   Param_163.WT7 := 2.050160e-01;
   Param_163.WT8 := 1.645390e-01;
   Param_164.WT1 := 1.000000e+00;
   Param_164.WT2 := 1.000000e+00;
   Param_164.WT3 := 6.709020e-02;
   Param_291.WT1 := 1.000000e+00;
   Param_291.WT2 := 1.000000e+00;
   Param_291.WT3 := 1.000000e+00;
   Param_291.WT4 := 1.000000e+00;
   Param_291.WT5 := 1.000000e+00;
   Param_291.WT6 := 1.000000e+00;
   Param_291.WT7 := 1.000000e+00;
   Param_291.WT8 := 1.000000e+00;
   Param_292.WT1 := 1.000000e+00;
   Param_292.WT2 := 1.000000e+00;
   Param_292.WT3 := 1.000000e+00;
   Param_292.WT4 := 1.000000e+00;
   Param_292.WT5 := 1.000000e+00;
   Param_292.WT6 := 1.000000e+00;
   Param_292.WT7 := 1.000000e+00;
   Param_292.WT8 := 1.000000e+00;
END_DATA_BLOCK

DATA_BLOCK "AIN_VALs_TEMP_661"	// DB 28
AUTHOR : RJ
VERSION : 0.1
"AIN"
BEGIN
END_DATA_BLOCK

DATA_BLOCK "AIN_VALs_PRESS_760"	// DB 29
AUTHOR : RJ
VERSION : 0.1
"AIN"
BEGIN
END_DATA_BLOCK

DATA_BLOCK "RESETSUM_VALs"	// DB 30
AUTHOR : RJ
VERSION : 0.1
  STRUCT
   Param_129 : UDT 25;	//Sheet 6 (RSM)
   Param_271 : UDT 25;	//Sheet 6 (RSM)
   Param_317 : UDT 25;	//Sheet 6 (RSM)
   Param_125 : UDT 25;	//Sheet 6 (RSM)
   Param_136 : UDT 25;	//Sheet 8 (RSM)
  END_STRUCT ;	
BEGIN
   Param_129.GAIN := 1.000000e+03;
   Param_271.GAIN := 1.000000e+00;
   Param_317.RCNT := 2.000000e+00;
   Param_317.GAIN := 1.000000e+00;
   Param_125.GAIN := 1.000000e+00;
   Param_136.GAIN := 1.000000e+00;
END_DATA_BLOCK

DATA_BLOCK "AIN_VALs_POS_25"	// DB 31
AUTHOR : RJ
VERSION : 0.1
"AIN"
BEGIN
END_DATA_BLOCK

DATA_BLOCK "XMULT_VALs"	// DB 32
AUTHOR : RJ
VERSION : 0.1
  STRUCT
   Param_X131 : UDT 26;	//Sheet 18 (RSM)
  END_STRUCT ;	
BEGIN
   Param_X131.PV_GAIN := 1.697100e-03;
   Param_X131.CAS_GAIN := 1.697000e-03;
   Param_X131.SCALE_TOP := 1.600000e+07;
   Param_X131.SCALE_BOT := -9.999900e+04;
END_DATA_BLOCK

DATA_BLOCK "ATCTime_VALs"	// DB 33
AUTHOR : RJ
FAMILY : ATC
VERSION : 0.1
  STRUCT
   T5OFF : S5TIME  := S5T#1S500MS;	//Sheet 2 (ATC)
   T6ON : S5TIME  := S5T#5M;	//Sheet 21 (ATC)
   T7ON : S5TIME  := S5T#10M30S;	//Sheet 22 (ATC)
   T8PULSE : S5TIME ;	//Sheet 28 (ATC)
   T9PULSE : S5TIME ;	//Sheet 30 (ATC)
   T10ON : S5TIME ;	//Sheet 45 (ATC)
  END_STRUCT ;	
BEGIN
END_DATA_BLOCK

DATA_BLOCK "DIGCNTNF_VALs"	// DB 34
AUTHOR : RJ
VERSION : 0.1
  STRUCT
   Param_036 : UDT 27;	//Sheet 3 (ATC)
  END_STRUCT ;	
BEGIN
   Param_036.N := 10;
END_DATA_BLOCK

DATA_BLOCK "Constants_ATC"	// DB 35
AUTHOR : RJ
FAMILY : ATC
VERSION : 0.1
  STRUCT
   FAIL13V : BOOL ;	//Sheet 5 (ATC)
   DIOBOK : BOOL  := TRUE;	//Sheet 5 (ATC)
   P06M17 : BOOL ;	//Sheet 28 (ATC)
   SYNCSPEED : REAL ;	//Sheet 48 (ATC)
  END_STRUCT ;	
BEGIN
END_DATA_BLOCK

DATA_BLOCK "RUNAVG_VALs_235"	// DB 36
AUTHOR : RJ
FAMILY : ATC
VERSION : 0.1
"RUNAVG"
BEGIN
END_DATA_BLOCK

DATA_BLOCK "AIN_VALs_POS_2"	// DB 37
AUTHOR : RJ
VERSION : 0.1
"AIN"
BEGIN
END_DATA_BLOCK

DATA_BLOCK "RSMTime_VALs"	// DB 38
AUTHOR : RJ
FAMILY : RSM
VERSION : 0.1
  STRUCT
   T1ON : S5TIME  := S5T#10S;	//Sheet 25 (RSM)
   T2PULSE : S5TIME  := S5T#1S;	//Sheet 27 (RSM)
   T3PULSE : S5TIME  := S5T#1S;	//Sheet 27 (RSM)
   T4OFF : S5TIME  := S5T#3M;	//Sheet 35 (RSM)
  END_STRUCT ;	
BEGIN
END_DATA_BLOCK

DATA_BLOCK "TIMECHG_VALs"	// DB 39
AUTHOR : RJ
VERSION : 0.1
  STRUCT
   Param_787 : UDT 28;	//Sheet 24 (ATC)
  END_STRUCT ;	
BEGIN
END_DATA_BLOCK

ORGANIZATION_BLOCK "Main program routine"	// OB 1
TITLE = "Main Program Sweep (Cycle)"
//Logic implementation of RSM & ATC, where each function call represents a single 
//sheet
//
AUTHOR : RJ
FAMILY : RSM,ATC
VERSION : 0.1
VAR_TEMP
  OB1_EV_CLASS : BYTE ;	//Bits 0-3 = 1 (Coming event), Bits 4-7 = 1 (Event class 1)
  OB1_SCAN_1 : BYTE ;	//1 (Cold restart scan 1 of OB 1), 3 (Scan 2-n of OB 1)
  OB1_PRIORITY : BYTE ;	//Priority of OB Execution
  OB1_OB_NUMBR : BYTE ;	//1 (Organization block 1, OB1)
  OB1_RESERVED_1 : BYTE ;	//Reserved for system
  OB1_RESERVED_2 : BYTE ;	//Reserved for system
  OB1_PREV_CYCLE : INT ;	//Cycle time of previous OB1 scan (milliseconds)
  OB1_MIN_CYCLE : INT ;	//Minimum cycle time of OB1 (milliseconds)
  OB1_MAX_CYCLE : INT ;	//Maximum cycle time of OB1 (milliseconds)
  OB1_DATE_TIME : DATE_AND_TIME ;	//Date and time OB1 started
END_VAR
BEGIN
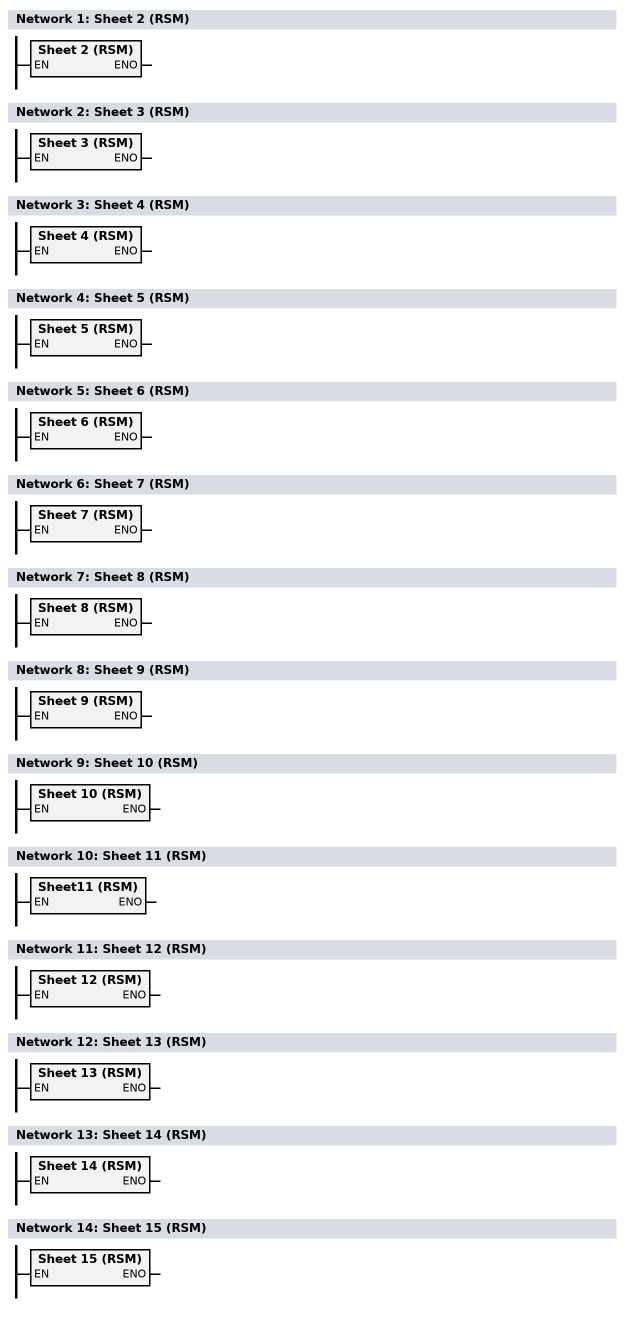
NETWORK
TITLE = Sheet 2 (RSM)
      CALL  "Sheet 2 (RSM)";
      NOP   0;
NETWORK
TITLE = Sheet 3 (RSM)
      CALL  "Sheet 3 (RSM)";
      NOP   0;
NETWORK
TITLE = Sheet 4 (RSM)
      CALL  "Sheet 4 (RSM)";
      NOP   0;
NETWORK
TITLE = Sheet 5 (RSM)
      CALL  "Sheet 5 (RSM)";
      NOP   0;
NETWORK
TITLE = Sheet 6 (RSM)
      CALL  "Sheet 6 (RSM)";
      NOP   0;
NETWORK
TITLE = Sheet 7 (RSM)
      CALL  "Sheet 7 (RSM)";
      NOP   0;
NETWORK
TITLE = Sheet 8 (RSM)
      CALL  "Sheet 8 (RSM)";
      NOP   0;
NETWORK
TITLE = Sheet 9 (RSM)
      CALL  "Sheet 9 (RSM)";
      NOP   0;
NETWORK
TITLE = Sheet 10 (RSM)
      CALL  "Sheet 10 (RSM)";
      NOP   0;
NETWORK
TITLE = Sheet 11 (RSM)
      CALL  "Sheet11 (RSM)";
      NOP   0;
NETWORK
TITLE = Sheet 12 (RSM)
      CALL  "Sheet 12 (RSM)";
      NOP   0;
NETWORK
TITLE = Sheet 13 (RSM)
      CALL  "Sheet 13 (RSM)";
      NOP   0;
NETWORK
TITLE = Sheet 14 (RSM)
      CALL  "Sheet 14 (RSM)";
      NOP   0;
NETWORK
TITLE = Sheet 15 (RSM)
      CALL  "Sheet 15 (RSM)";
      NOP   0;
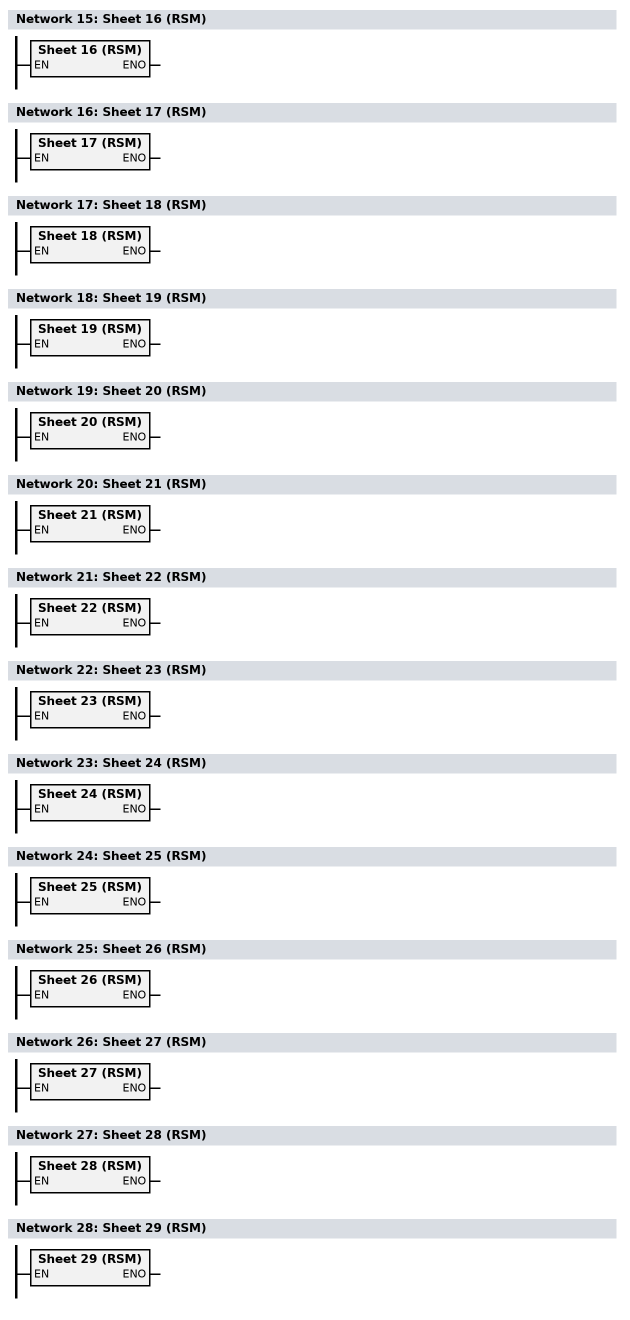
NETWORK
TITLE = Sheet 16 (RSM)
      CALL  "Sheet 16 (RSM)";
      NOP   0;
NETWORK
TITLE = Sheet 17 (RSM)
      CALL  "Sheet 17 (RSM)";
      NOP   0;
NETWORK
TITLE = Sheet 18 (RSM)
      CALL  "Sheet 18 (RSM)";
      NOP   0;
NETWORK
TITLE = Sheet 19 (RSM)
      CALL  "Sheet 19 (RSM)";
      NOP   0;
NETWORK
TITLE = Sheet 20 (RSM)
      CALL  "Sheet 20 (RSM)";
      NOP   0;
NETWORK
TITLE = Sheet 21 (RSM)
      CALL  "Sheet 21 (RSM)";
      NOP   0;
NETWORK
TITLE = Sheet 22 (RSM)
      CALL  "Sheet 22 (RSM)";
      NOP   0;
NETWORK
TITLE = Sheet 23 (RSM)
      CALL  "Sheet 23 (RSM)";
      NOP   0;
NETWORK
TITLE = Sheet 24 (RSM)
      CALL  "Sheet 24 (RSM)";
      NOP   0;
NETWORK
TITLE = Sheet 25 (RSM)
      CALL  "Sheet 25 (RSM)";
      NOP   0;
NETWORK
TITLE = Sheet 26 (RSM)
      CALL  "Sheet 26 (RSM)";
      NOP   0;
NETWORK
TITLE = Sheet 27 (RSM)
      CALL  "Sheet 27 (RSM)";
      NOP   0;
NETWORK
TITLE = Sheet 28 (RSM)
      CALL  "Sheet 28 (RSM)";
      NOP   0;
NETWORK
TITLE = Sheet 29 (RSM)
      CALL  "Sheet 29 (RSM)";
      NOP   0;
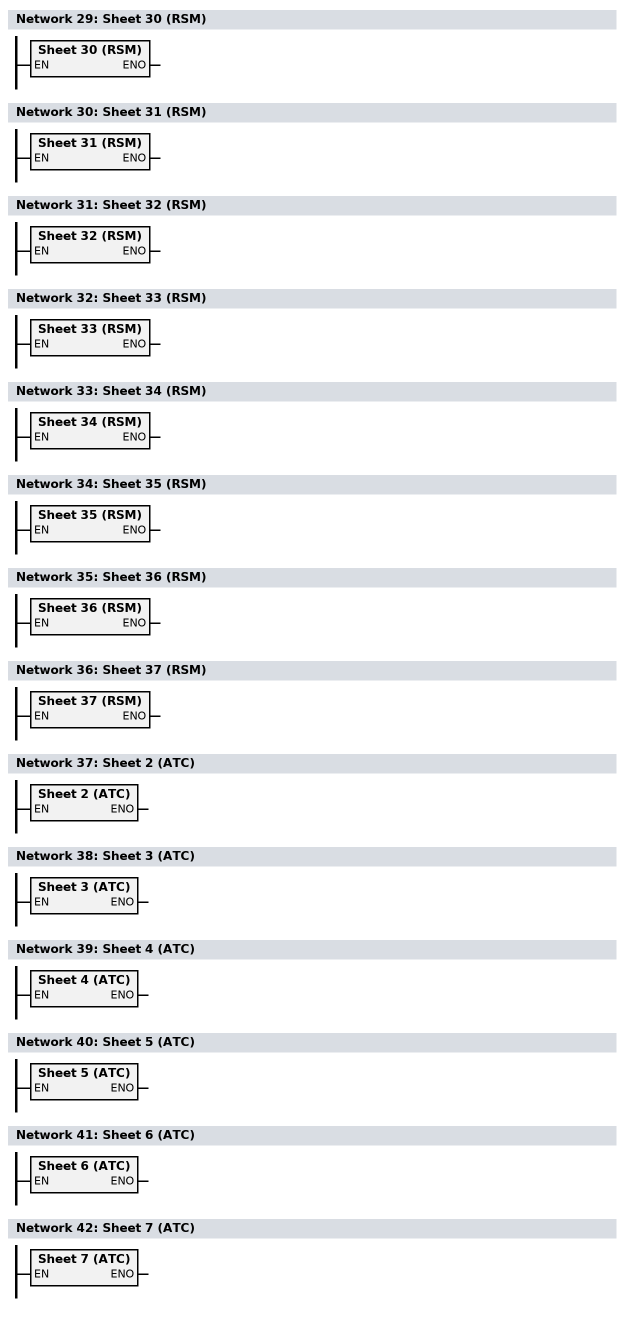
NETWORK
TITLE = Sheet 30 (RSM)
      CALL  "Sheet 30 (RSM)";
      NOP   0;
NETWORK
TITLE = Sheet 31 (RSM)
      CALL  "Sheet 31 (RSM)";
      NOP   0;
NETWORK
TITLE = Sheet 32 (RSM)
      CALL  "Sheet 32 (RSM)";
      NOP   0;
NETWORK
TITLE = Sheet 33 (RSM)
      CALL  "Sheet 33 (RSM)";
      NOP   0;
NETWORK
TITLE = Sheet 34 (RSM)
      CALL  "Sheet 34 (RSM)";
      NOP   0;
NETWORK
TITLE = Sheet 35 (RSM)
      CALL  "Sheet 35 (RSM)";
      NOP   0;
NETWORK
TITLE = Sheet 36 (RSM)
      CALL  "Sheet 36 (RSM)";
      NOP   0;
NETWORK
TITLE = Sheet 37 (RSM)
      CALL  "Sheet 37 (RSM)";
      NOP   0;
NETWORK
TITLE = Sheet 2 (ATC)
      CALL  "Sheet 2 (ATC)";
      NOP   0;
NETWORK
TITLE = Sheet 3 (ATC)
      CALL  "Sheet 3 (ATC)";
      NOP   0;
NETWORK
TITLE = Sheet 4 (ATC)
      CALL  "Sheet 4 (ATC)";
      NOP   0;
NETWORK
TITLE = Sheet 5 (ATC)
      CALL  "Sheet 5 (ATC)";
      NOP   0;
NETWORK
TITLE = Sheet 6 (ATC)
      CALL  "Sheet 6 (ATC)";
      NOP   0;
NETWORK
TITLE = Sheet 7 (ATC)
      CALL  "Sheet 7 (ATC)";
      NOP   0;
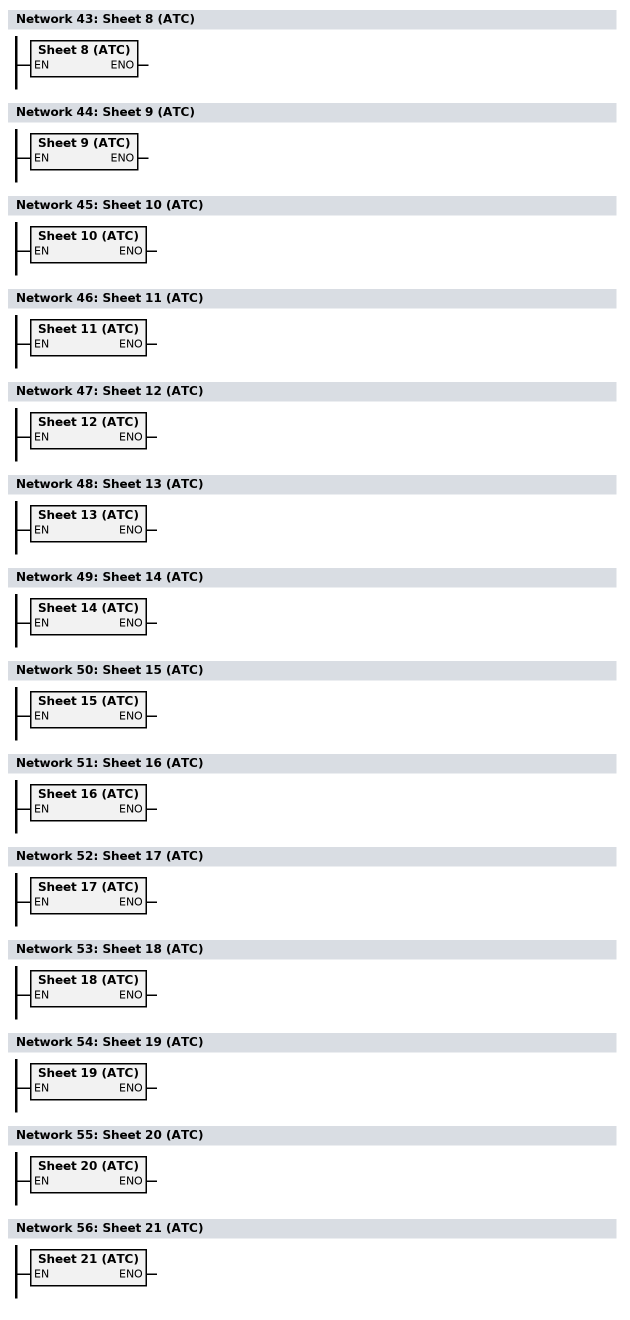
NETWORK
TITLE = Sheet 8 (ATC)
      CALL  "Sheet 8 (ATC)";
      NOP   0;
NETWORK
TITLE = Sheet 9 (ATC)
      CALL  "Sheet 9 (ATC)";
      NOP   0;
NETWORK
TITLE = Sheet 10 (ATC)
      CALL  "Sheet 10 (ATC)";
      NOP   0;
NETWORK
TITLE = Sheet 11 (ATC)
      CALL  "Sheet 11 (ATC)";
      NOP   0;
NETWORK
TITLE = Sheet 12 (ATC)
      CALL  "Sheet 12 (ATC)";
      NOP   0;
NETWORK
TITLE = Sheet 13 (ATC)
      CALL  "Sheet 13 (ATC)";
      NOP   0;
NETWORK
TITLE = Sheet 14 (ATC)
      CALL  "Sheet 14 (ATC)";
      NOP   0;
NETWORK
TITLE = Sheet 15 (ATC)
      CALL  "Sheet 15 (ATC)";
      NOP   0;
NETWORK
TITLE = Sheet 16 (ATC)
      CALL  "Sheet 16 (ATC)";
      NOP   0;
NETWORK
TITLE = Sheet 17 (ATC)
      CALL  "Sheet 17 (ATC)";
      NOP   0;
NETWORK
TITLE = Sheet 18 (ATC)
      CALL  "Sheet 18 (ATC)";
      NOP   0;
NETWORK
TITLE = Sheet 19 (ATC)
      CALL  "Sheet 19 (ATC)";
      NOP   0;
NETWORK
TITLE = Sheet 20 (ATC)
      CALL  "Sheet 20 (ATC)";
      NOP   0;
NETWORK
TITLE = Sheet 21 (ATC)
      CALL  "Sheet 21 (ATC)";
      NOP   0;
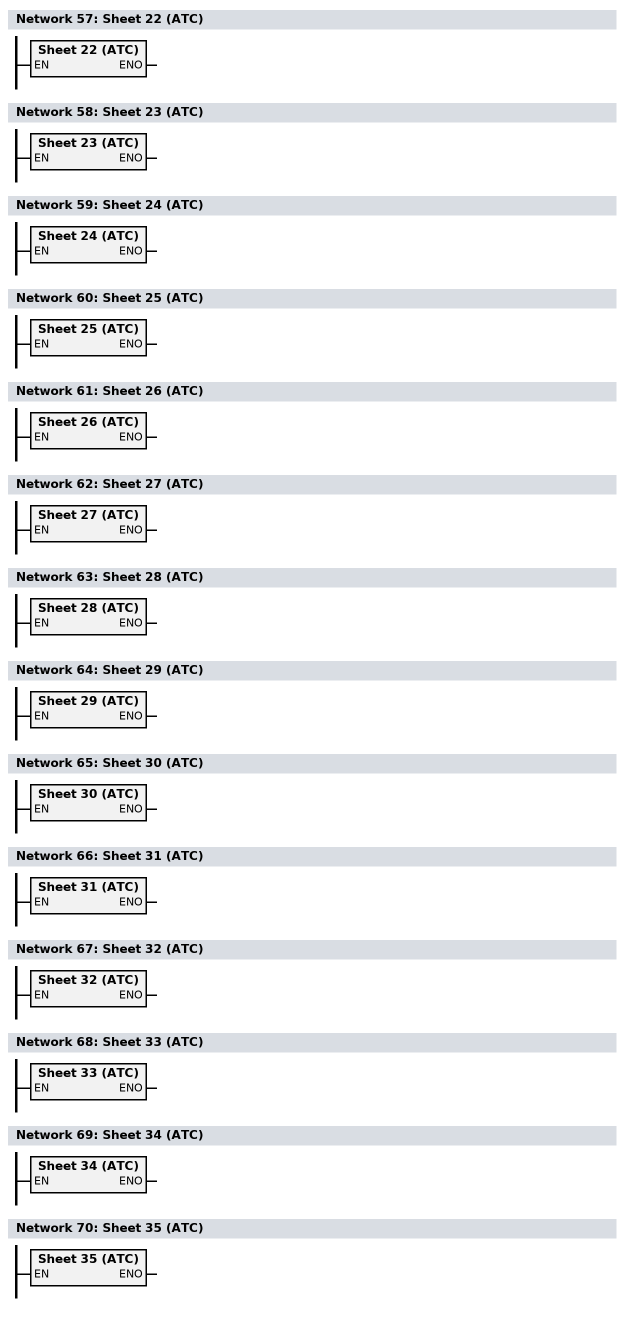
NETWORK
TITLE = Sheet 22 (ATC)
      CALL  "Sheet 22 (ATC)";
      NOP   0;
NETWORK
TITLE = Sheet 23 (ATC)
      CALL  "Sheet 23 (ATC)";
      NOP   0;
NETWORK
TITLE = Sheet 24 (ATC)
      CALL  "Sheet 24 (ATC)";
      NOP   0;
NETWORK
TITLE = Sheet 25 (ATC)
      CALL  "Sheet 25 (ATC)";
      NOP   0;
NETWORK
TITLE = Sheet 26 (ATC)
      CALL  "Sheet 26 (ATC)";
      NOP   0;
NETWORK
TITLE = Sheet 27 (ATC)
      CALL  "Sheet 27 (ATC)";
      NOP   0;
NETWORK
TITLE = Sheet 28 (ATC)
      CALL  "Sheet 28 (ATC)";
      NOP   0;
NETWORK
TITLE = Sheet 29 (ATC)
      CALL  "Sheet 29 (ATC)";
      NOP   0;
NETWORK
TITLE = Sheet 30 (ATC)
      CALL  "Sheet 30 (ATC)";
      NOP   0;
NETWORK
TITLE = Sheet 31 (ATC)
      CALL  "Sheet 31 (ATC)";
      NOP   0;
NETWORK
TITLE = Sheet 32 (ATC)
      CALL  "Sheet 32 (ATC)";
      NOP   0;
NETWORK
TITLE = Sheet 33 (ATC)
      CALL  "Sheet 33 (ATC)";
      NOP   0;
NETWORK
TITLE = Sheet 34 (ATC)
      CALL  "Sheet 34 (ATC)";
      NOP   0;
NETWORK
TITLE = Sheet 35 (ATC)
      CALL  "Sheet 35 (ATC)";
      NOP   0;
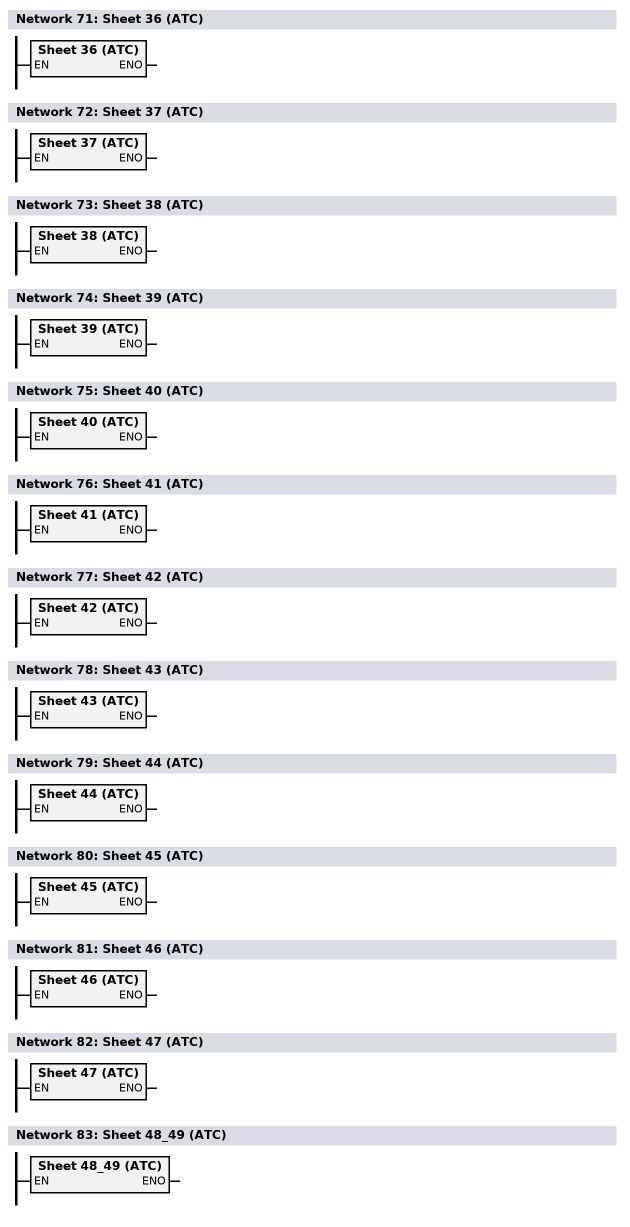
NETWORK
TITLE = Sheet 36 (ATC)
      CALL  "Sheet 36 (ATC)";
      NOP   0;
NETWORK
TITLE = Sheet 37 (ATC)
      CALL  "Sheet 37 (ATC)";
      NOP   0;
NETWORK
TITLE = Sheet 38 (ATC)
      CALL  "Sheet 38 (ATC)";
      NOP   0;
NETWORK
TITLE = Sheet 39 (ATC)
      CALL  "Sheet 39 (ATC)";
      NOP   0;
NETWORK
TITLE = Sheet 40 (ATC)
      CALL  "Sheet 40 (ATC)";
      NOP   0;
NETWORK
TITLE = Sheet 41 (ATC)
      CALL  "Sheet 41 (ATC)";
      NOP   0;
NETWORK
TITLE = Sheet 42 (ATC)
      CALL  "Sheet 42 (ATC)";
      NOP   0;
NETWORK
TITLE = Sheet 43 (ATC)
      CALL  "Sheet 43 (ATC)";
      NOP   0;
NETWORK
TITLE = Sheet 44 (ATC)
      CALL  "Sheet 44 (ATC)";
      NOP   0;
NETWORK
TITLE = Sheet 45 (ATC)
      CALL  "Sheet 45 (ATC)";
      NOP   0;
NETWORK
TITLE = Sheet 46 (ATC) 
      CALL  "Sheet 46 (ATC)";
      NOP   0;
NETWORK
TITLE = Sheet 47 (ATC)
      CALL  "Sheet 47 (ATC)";
      NOP   0;
NETWORK
TITLE = Sheet 48_49 (ATC)
      CALL  "Sheet 48_49 (ATC)";
      NOP   0;
END_ORGANIZATION_BLOCK

ORGANIZATION_BLOCK "I/O_FLT1"	// OB 82
TITLE = "I/O Point Fault"
AUTHOR : RJ
VERSION : 0.1
VAR_TEMP
  OB82_EV_CLASS : BYTE ;	//16#39, Event class 3, Entering event state, Internal fault event
  OB82_FLT_ID : BYTE ;	//16#XX, Fault identifcation code
  OB82_PRIORITY : BYTE ;	//Priority of OB Execution
  OB82_OB_NUMBR : BYTE ;	//82 (Organization block 82, OB82)
  OB82_RESERVED_1 : BYTE ;	//Reserved for system
  OB82_IO_FLAG : BYTE ;	//Input (01010100), Output (01010101)
  OB82_MDL_ADDR : WORD ;	//Base address of module with fault
  OB82_MDL_DEFECT : BOOL ;	//Module defective
  OB82_INT_FAULT : BOOL ;	//Internal fault
  OB82_EXT_FAULT : BOOL ;	//External fault
  OB82_PNT_INFO : BOOL ;	//Point information
  OB82_EXT_VOLTAGE : BOOL ;	//External voltage low
  OB82_FLD_CONNCTR : BOOL ;	//Field wiring connector missing
  OB82_NO_CONFIG : BOOL ;	//Module has no configuration data
  OB82_CONFIG_ERR : BOOL ;	//Module has configuration error
  OB82_MDL_TYPE : BYTE ;	//Type of module
  OB82_SUB_MDL_ERR : BOOL ;	//Sub-Module is missing or has error
  OB82_COMM_FAULT : BOOL ;	//Communication fault
  OB82_MDL_STOP : BOOL ;	//Module is stopped
  OB82_WTCH_DOG_FLT : BOOL ;	//Watch dog timer stopped module
  OB82_INT_PS_FLT : BOOL ;	//Internal power supply fault
  OB82_PRIM_BATT_FLT : BOOL ;	//Primary battery is in fault
  OB82_BCKUP_BATT_FLT : BOOL ;	//Backup battery is in fault
  OB82_RESERVED_2 : BOOL ;	//Reserved for system
  OB82_RACK_FLT : BOOL ;	//Rack fault, only for bus interface module
  OB82_PROC_FLT : BOOL ;	//Processor fault
  OB82_EPROM_FLT : BOOL ;	//EPROM fault
  OB82_RAM_FLT : BOOL ;	//RAM fault
  OB82_ADU_FLT : BOOL ;	//ADU fault
  OB82_FUSE_FLT : BOOL ;	//Fuse fault
  OB82_HW_INTR_FLT : BOOL ;	//Hardware interupt input in fault
  OB82_RESERVED_3 : BOOL ;	//Reserved for system
  OB82_DATE_TIME : DATE_AND_TIME ;	//Date and time OB82 started
END_VAR
BEGIN
// (block stored without names or comments; labels and parameter names are numbered)
END_ORGANIZATION_BLOCK

ORGANIZATION_BLOCK "I/O_FLT2"	// OB 83
TITLE = "I/O Point Fault"
AUTHOR : RJ
VERSION : 0.1
VAR_TEMP
  OB83_EV_CLASS : BYTE ;	//16#38/39, Event class 3, module inserted/removed (8/9)
  OB83_FLT_ID : BYTE ;	//16#XX, Fault identifcation code
  OB83_PRIORITY : BYTE ;	//Priority of OB Execution
  OB83_OB_NUMBR : BYTE ;	//83 (Organization block 83, OB83)
  OB83_RESERVED_1 : BYTE ;	//Reserved for system
  OB83_MDL_ID : BYTE ;	//Input module (01010100), Output module (01010101)
  OB83_MDL_ADDR : WORD ;	//Base address of module with point fault
  OB83_RACK_NUM : INT ;	//Number of rack that has module with point fault
  OB83_MDL_TYPE : WORD ;	//Module type with point fault
  OB83_DATE_TIME : DATE_AND_TIME ;	//Date and time OB83 started
END_VAR
BEGIN
// (block stored without names or comments; labels and parameter names are numbered)
END_ORGANIZATION_BLOCK

ORGANIZATION_BLOCK "OBNL_FLT"	// OB 85
TITLE = "Organization Block (OB) Not Loaded Fault"
AUTHOR : RJ
VERSION : 0.1
VAR_TEMP
  OB85_EV_CLASS : BYTE ;	//16#35 Event class 3
  OB85_FLT_ID : BYTE ;	//16#XX, Fault identification code
  OB85_PRIORITY : BYTE ;	//Priority of OB Execution
  OB85_OB_NUMBR : BYTE ;	//85 (Organization block 85, OB85)
  OB85_RESERVED_1 : BYTE ;	//Reserved for system
  OB85_RESERVED_2 : BYTE ;	//Reserved for system
  OB85_RESERVED_3 : INT ;	//Reserved for system
  OB85_ERR_EV_CLASS : BYTE ;	//Class of event causing error
  OB85_ERR_EV_NUM : BYTE ;	//Number of event causing error
  OB85_OB_PRIOR : BYTE ;	//Priority of OB causing error
  OB85_OB_NUM : BYTE ;	//Number of OB causing error
  OB85_DATE_TIME : DATE_AND_TIME ;	//Date and time OB85 started
END_VAR
BEGIN
// (block stored without names or comments; labels and parameter names are numbered)
END_ORGANIZATION_BLOCK

ORGANIZATION_BLOCK "RACK_FLT"	// OB 86
TITLE = "Loss Of Rack Fault"
AUTHOR : RJ
VERSION : 0.1
VAR_TEMP
  OB86_EV_CLASS : BYTE ;	//16#38/39 Event class 3
  OB86_FLT_ID : BYTE ;	//16#C1/C4/C5, Fault identifcation code
  OB86_PRIORITY : BYTE ;	//Priority of OB Execution
  OB86_OB_NUMBR : BYTE ;	//86 (Organization block 86, OB86)
  OB86_RESERVED_1 : BYTE ;	//Reserved for system
  OB86_RESERVED_2 : BYTE ;	//Reserved for system
  OB86_MDL_ADDR : WORD ;	//Base address of IM module in rack with fault
  OB86_RACKS_FLTD : ARRAY  [0 .. 31 ] OF BOOL ;	//Racks in fault
  OB86_DATE_TIME : DATE_AND_TIME ;	//Date and time OB86 started
END_VAR
BEGIN
// (block stored without names or comments; labels and parameter names are numbered)
END_ORGANIZATION_BLOCK

ORGANIZATION_BLOCK "COMPLETE RESTART"	// OB 100
TITLE = "Complete Restart"
VERSION : 0.1
VAR_TEMP
  OB100_EV_CLASS : BYTE ;	//16#13, Event class 1, Entering event state, Event logged in diagnostic buffer
  OB100_STRTUP : BYTE ;	//16#81/82/83/84 Method of startup
  OB100_PRIORITY : BYTE ;	//Priority of OB Execution
  OB100_OB_NUMBR : BYTE ;	//100 (Organization block 100, OB100)
  OB100_RESERVED_1 : BYTE ;	//Reserved for system
  OB100_RESERVED_2 : BYTE ;	//Reserved for system
  OB100_STOP : WORD ;	//Event that caused CPU to stop (16#4xxx)
  OB100_STRT_INFO : DWORD ;	//Information on how system started
  OB100_DATE_TIME : DATE_AND_TIME ;	//Date and time OB100 started
  RET : INT ;
  CDT : DATE_AND_TIME ;
  CTime : TIME_OF_DAY ;
END_VAR
BEGIN
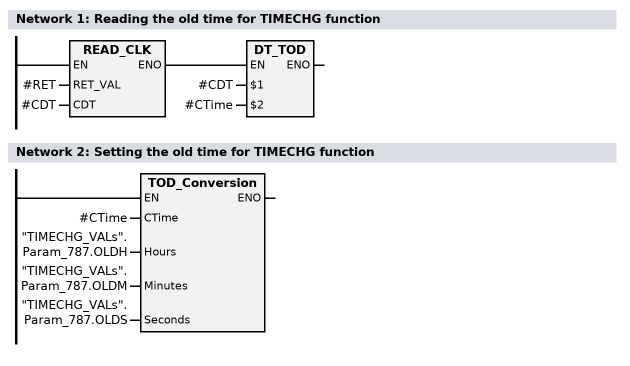
NETWORK
TITLE = Reading the old time for TIMECHG function
      A(;
      CALL  "READ_CLK" (
           RET_VAL                  := #RET,
           CDT                      := #CDT);
      A     BR;
      );
      JNB   _001;
      CALL  "DT_TOD" (
           $1                       := #CDT,
           $2                       := #CTime);
_001: NOP   0;
NETWORK
TITLE = Setting the old time for TIMECHG function
      CALL  "TOD_Conversion" (
           CTime                    := #CTime,
           Hours                    := "TIMECHG_VALs".Param_787.OLDH,
           Minutes                  := "TIMECHG_VALs".Param_787.OLDM,
           Seconds                  := "TIMECHG_VALs".Param_787.OLDS);
      NOP   0;
END_ORGANIZATION_BLOCK

ORGANIZATION_BLOCK "PROG_ERR"	// OB 121
TITLE = "Programming Error"
AUTHOR : RJ
VERSION : 0.1
VAR_TEMP
  OB121_EV_CLASS : BYTE ;	//16#25, Event class 2, Entering event state, Internal fault event
  OB121_SW_FLT : BYTE ;	//16#XX Software programming fault
  OB121_PRIORITY : BYTE ;	//Priority of OB Execution
  OB121_OB_NUMBR : BYTE ;	//121 (Organization block 121, OB121)
  OB121_BLK_TYPE : BYTE ;	//16#88/8A/8B/8C/8E Type of block fault occured in
  OB121_RESERVED_1 : BYTE ;	//Reserved for system
  OB121_FLT_REG : WORD ;	//16#XX Specific register that caused fault
  OB121_BLK_NUM : WORD ;	//Number of block that programming fault occured in
  OB121_PRG_ADDR : WORD ;	//Address in block where programming fault occured
  OB121_DATE_TIME : DATE_AND_TIME ;	//Date and time OB121 started
END_VAR
BEGIN
// (block stored without names or comments; labels and parameter names are numbered)
END_ORGANIZATION_BLOCK

ORGANIZATION_BLOCK "MOD_ERR"	// OB 122
TITLE = "Module Access Error"
AUTHOR : RJ
VERSION : 0.1
VAR_TEMP
  OB122_EV_CLASS : BYTE ;	//16#29, Event class 2, Entering event state, Internal fault event
  OB122_SW_FLT : BYTE ;	//16#XX Software error code
  OB122_PRIORITY : BYTE ;	//Priority of OB Execution
  OB122_OB_NUMBR : BYTE ;	//122 (Organization block 122, OB122)
  OB122_BLK_TYPE : BYTE ;	//16#88/8C/8E Type of block fault occured in
  OB122_MEM_AREA : BYTE ;	//Memory area where access error occured
  OB122_MEM_ADDR : WORD ;	//Memory address where access error occured
  OB122_BLK_NUM : WORD ;	//Block number in which error occured
  OB122_PRG_ADDR : WORD ;	//Program address where error occured
  OB122_DATE_TIME : DATE_AND_TIME ;	//Date and time OB1 started
END_VAR
BEGIN
// (block stored without names or comments; labels and parameter names are numbered)
END_ORGANIZATION_BLOCK

SYMBOL_TABLE
"ASL1"	I 0.0	BOOL	// Auto Stop Latched # 1 (OPC) - (FieldIO1-M1)
"BR1"	I 0.1	BOOL	//  (OPC) - (FieldIO1-M1)
"INFV1"	I 0.2	BOOL	//  (OPC) - (FieldIO1-M1)
"TGRB1"	I 0.3	BOOL	//  (OPC) - (FieldIO1-M1)
"CSVBP"	I 0.4	BOOL	//  (OPC) - (FieldIO1-M1)
"CSVPB"	I 0.5	BOOL	//  (OPC) - (FieldIO1-M1)
"LCHPB"	I 0.6	BOOL	//  (OPC) - (FieldIO1-M1)
"LTPB"	I 0.7	BOOL	//  (OPC) - (FieldIO1-M1)
"OSVPB"	I 1.0	BOOL	//  (OPC) - (FieldIO1-M1)
"TMPB"	I 1.1	BOOL	//  (OPC) - (FieldIO1-M1)
"OPCT"	I 1.2	BOOL	//  (OPC) - (FieldIO1-M1)
"OST"	I 1.3	BOOL	//  (OPC) - (FieldIO1-M1)
"ADSDN"	I 2.0	BOOL	//  (OA) - (FieldIO1-M2)
"ADSPERM"	I 2.1	BOOL	//  (OA) - (FieldIO1-M2)
"ADSUP"	I 2.2	BOOL	//  (OA) - (FieldIO1-M2)
"VPLDN"	I 2.3	BOOL	//  (OA) - (FieldIO1-M2)
"VPLPERM"	I 2.4	BOOL	//  (OA) - (FieldIO1-M2)
"VPLUP"	I 2.5	BOOL	//  (OA) - (FieldIO1-M2)
"ASDN"	I 2.6	BOOL	//  (OA) - (FieldIO1-M2)
"ASPERM"	I 2.7	BOOL	//  (OA) - (FieldIO1-M2)
"ASUP"	I 3.0	BOOL	//  (OA) - (FieldIO1-M2)
"CDLPERM"	I 3.1	BOOL	//  (OA) - (FieldIO1-M2)
"FL13PRI"	I 3.2	BOOL	//  (OA) - (FieldIO1-M2)
"FL13STY"	I 3.3	BOOL	//  (OA) - (FieldIO1-M2)
"FLOACPRI"	I 3.4	BOOL	//  (OA) - (FieldIO1-M2)
"FLOACSTY"	I 3.5	BOOL	//  (OA) - (FieldIO1-M2)
"FLOPCPRI"	I 3.6	BOOL	//  (OA) - (FieldIO1-M2)
"FLOPCSTY"	I 3.7	BOOL	//  (OA) - (FieldIO1-M2)
"ASL2"	I 4.0	BOOL	//  (OPC) - (FieldIO2-M1)
"BR2"	I 4.1	BOOL	//  (OPC) - (FieldIO2-M1)
"INFV2"	I 4.2	BOOL	//  (OPC) - (FieldIO2-M1)
"TGRB2"	I 4.3	BOOL	//  (OPC) - (FieldIO2-M1)
"IV1CL"	I 6.0	BOOL	//  (OA) - (FieldIO2-M2)
"IV1OP"	I 6.1	BOOL	//  (OA) - (FieldIO2-M2)
"IV2CL"	I 6.2	BOOL	//  (OA) - (FieldIO2-M2)
"IV2OP"	I 6.3	BOOL	//  (OA) - (FieldIO2-M2)
"IV3CL"	I 6.4	BOOL	//  (OA) - (FieldIO2-M2)
"IV3OP"	I 6.5	BOOL	//  (OA) - (FieldIO2-M2)
"IV4CL"	I 6.6	BOOL	//  (OA) - (FieldIO2-M2)
"IV4OP"	I 6.7	BOOL	//  (OA) - (FieldIO2-M2)
"RV1CL"	I 7.0	BOOL	//  (OA) - (FieldIO2-M2)
"RV1OP"	I 7.1	BOOL	//  (OA) - (FieldIO2-M2)
"RV2CL"	I 7.2	BOOL	//  (OA) - (FieldIO2-M2)
"RV2OP"	I 7.3	BOOL	//  (OA) - (FieldIO2-M2)
"RV3CL"	I 7.4	BOOL	//  (OA) - (FieldIO2-M2)
"RV3OP"	I 7.5	BOOL	//  (OA) - (FieldIO2-M2)
"RV4CL"	I 7.6	BOOL	//  (OA) - (FieldIO2-M2)
"RV4OP"	I 7.7	BOOL	//  (OA) - (FieldIO2-M2)
"ASL3"	I 8.0	BOOL	//  (OPC) - (FieldIO3-M1)
"BR3"	I 8.1	BOOL	//  (OPC) - (FieldIO3-M1)
"INFV3"	I 8.2	BOOL	//  (OPC) - (FieldIO3-M1)
"TGRB3"	I 8.3	BOOL	//  (OPC) - (FieldIO3-M1)
"MSVLC"	I 8.4	BOOL	//  (OPC) - (FieldIO3-M1)
"MSVLO"	I 8.5	BOOL	//  (OPC) - (FieldIO3-M1)
"MSVRC"	I 8.6	BOOL	//  (OPC) - (FieldIO3-M1)
"MSVRO"	I 8.7	BOOL	//  (OPC) - (FieldIO3-M1)
"CI0284"	I 9.0	BOOL	//  (OPC) - (FieldIO3-M1)
"SRVOIN"	I 9.1	BOOL	//  (OPC) - (FieldIO3-M1)
"BCIV"	I 9.2	BOOL	//  (OPC) - (FieldIO3-M1)
"HOLDLOAD"	I 10.0	BOOL	//  (OA) - (FieldIO3-M2)
"REJIMP"	I 10.1	BOOL	//  (OA) - (FieldIO3-M2)
"REJMW"	I 10.2	BOOL	//  (OA) - (FieldIO3-M2)
"RESETADS"	I 10.3	BOOL	//  (OA) - (FieldIO3-M2)
"MWA"	IW 512	WORD	//  (OPC) - (FieldIO1-M5)
"OPSA"	IW 514	WORD	//  (OPC) - (FieldIO1-M5)
"OPXA"	IW 516	WORD	//  (OPC) - (FieldIO1-M5)
"TPA"	IW 518	WORD	//  (OPC) - (FieldIO1-M5)
"PIA"	IW 520	WORD	//  (OA) - (FieldIO1-M5)
"GSH1"	IW 522	WORD	//  (OA) - (FieldIO1-M5)
"STATCUR"	IW 524	WORD	//  (OPC) - (FieldIO1-M5)
"MWB"	IW 528	WORD	//  (OPC) - (FieldIO2-M5)
"OPSB"	IW 530	WORD	//  (OPC) - (FieldIO2-M5)
"OPXB"	IW 532	WORD	//  (OPC) - (FieldIO2-M5)
"TPB"	IW 534	WORD	//  (OPC) - (FieldIO2-M5)
"PIB"	IW 536	WORD	//  (OA) - (FieldIO2-M5)
"GSHP2"	IW 538	WORD	//  (OA) - (FieldIO2-M5)
"PLRL"	IW 540	WORD	//  (OA) - (FieldIO2-M5)
"MWC"	IW 544	WORD	//  (OPC) - (FieldIO3-M5)
"OPSC"	IW 546	WORD	//  (OPC) - (FieldIO3-M5)
"OPXC"	IW 548	WORD	//  (OPC) - (FieldIO3-M5)
"TPC"	IW 550	WORD	//  (OPC) - (FieldIO3-M5)
"PIC"	IW 552	WORD	//  (OA) - (FieldIO3-M5)
"MVAR"	IW 554	WORD	//  (OPC) - (FieldIO3-M5)
"OBNL_FLT"	OB 85	OB 85	// OB Not Loaded Fault
"PROG_ERR"	OB 121	OB 121	// Programming Error
"MOD_ERR"	OB 122	OB 122	// Module Access Error
"TM1"	Q 0.0	BOOL	//  (OPC) - (FieldIO1-M3)
"LATCH1"	Q 0.1	BOOL	//  (OPC) - (FieldIO1-M3)
"TTRIP1"	Q 0.2	BOOL	//  (OPC) - (FieldIO1-M3)
"PSMN1"	Q 0.3	BOOL	//  (OPC) - (FieldIO1-M3)
"OSPD1"	Q 0.4	BOOL	//  (OPC) - (FieldIO1-M3)
"SRVOOUT1"	Q 0.5	BOOL	//  (OPC) - (FieldIO1-M3)
"OPCO1"	Q 0.6	BOOL	//  (OPC) - (FieldIO1-M3)
"OPMN1"	Q 0.7	BOOL	//  (OPC) - (FieldIO1-M3)
"MRBC"	Q 1.0	BOOL	//  (OPC) - (FieldIO1-M3)
"MRBRC"	Q 1.1	BOOL	//  (OPC) - (FieldIO1-M3)
"MVPMAN"	Q 1.2	BOOL	//  (OPC) - (FieldIO1-M3)
"ASLNLT"	Q 1.3	BOOL	//  (OPC) - (FieldIO1-M3)
"ASLT"	Q 1.4	BOOL	//  (OPC) - (FieldIO1-M3)
"GVCL"	Q 1.5	BOOL	//  (OPC) - (FieldIO1-M3)
"LT"	Q 1.6	BOOL	//  (OPC) - (FieldIO1-M3)
"ADS1"	Q 2.0	BOOL	//  (OA) - (FieldIO1-M4)
"AS1"	Q 2.1	BOOL	//  (OA) - (FieldIO1-M4)
"BRCTT1"	Q 2.2	BOOL	//  (OA) - (FieldIO1-M4)
"DMWFL1"	Q 2.3	BOOL	//  (OA) - (FieldIO1-M4)
"HLLL1"	Q 2.4	BOOL	//  (OA) - (FieldIO1-M4)
"IPI1"	Q 2.5	BOOL	//  (OA) - (FieldIO1-M4)
"LLLL1"	Q 2.6	BOOL	//  (OA) - (FieldIO1-M4)
"LOWFRQ1"	Q 2.7	BOOL	//  (OA) - (FieldIO1-M4)
"MWFAIL1"	Q 3.0	BOOL	//  (OA) - (FieldIO1-M4)
"MWI1"	Q 3.1	BOOL	//  (OA) - (FieldIO1-M4)
"OA1"	Q 3.2	BOOL	//  (OA) - (FieldIO1-M4)
"OPXFAIL1"	Q 3.3	BOOL	//  (OA) - (FieldIO1-M4)
"PIFAIL1"	Q 3.4	BOOL	//  (OA) - (FieldIO1-M4)
"PLRLL1"	Q 3.5	BOOL	//  (OA) - (FieldIO1-M4)
"SPI1"	Q 3.6	BOOL	//  (OA) - (FieldIO1-M4)
"TPFAIL1"	Q 3.7	BOOL	//  (OA) - (FieldIO1-M4)
"TM2"	Q 4.0	BOOL	//  (OPC) - (FieldIO2-M3)
"LATCH2"	Q 4.1	BOOL	//  (OPC) - (FieldIO2-M3)
"TTRIP2"	Q 4.2	BOOL	//  (OPC) - (FieldIO2-M3)
"PSMN2"	Q 4.3	BOOL	//  (OPC) - (FieldIO2-M3)
"OSPD2"	Q 4.4	BOOL	//  (OPC) - (FieldIO2-M3)
"SRVOOUT2"	Q 4.5	BOOL	//  (OPC) - (FieldIO2-M3)
"OPCO2"	Q 4.6	BOOL	//  (OPC) - (FieldIO2-M3)
"OPMN2"	Q 4.7	BOOL	//  (OPC) - (FieldIO2-M3)
"MWLT"	Q 5.0	BOOL	//  (OPC) - (FieldIO2-M3)
"OPCMONLT"	Q 5.1	BOOL	//  (OPC) - (FieldIO2-M3)
"PFAILT"	Q 5.2	BOOL	//  (OPC) - (FieldIO2-M3)
"RPMLT"	Q 5.3	BOOL	//  (OPC) - (FieldIO2-M3)
"STROBE"	Q 5.4	BOOL	//  (OPC) - (FieldIO2-M3)
"TMLT"	Q 5.5	BOOL	//  (OPC) - (FieldIO2-M3)
"TMLT1"	Q 5.6	BOOL	//  (OPC) - (FieldIO2-M3)
"TVCL"	Q 5.7	BOOL	//  (OPC) - (FieldIO2-M3)
"ADS2"	Q 6.0	BOOL	//  (OA) - (FieldIO2-M4)
"AS2"	Q 6.1	BOOL	//  (OA) - (FieldIO2-M4)
"BRCTT2"	Q 6.2	BOOL	//  (OA) - (FieldIO2-M4)
"DMWFL2"	Q 6.3	BOOL	//  (OA) - (FieldIO2-M4)
"HLLL2"	Q 6.4	BOOL	//  (OA) - (FieldIO2-M4)
"IPI2"	Q 6.5	BOOL	//  (OA) - (FieldIO2-M4)
"LLLL2"	Q 6.6	BOOL	//  (OA) - (FieldIO2-M4)
"LOWFRQ2"	Q 6.7	BOOL	//  (OA) - (FieldIO2-M4)
"MWFAIL2"	Q 7.0	BOOL	//  (OA) - (FieldIO2-M4)
"MWI2"	Q 7.1	BOOL	//  (OA) - (FieldIO2-M4)
"OA2"	Q 7.2	BOOL	//  (OA) - (FieldIO2-M4)
"OPXFAIL2"	Q 7.3	BOOL	//  (OA) - (FieldIO2-M4)
"PIFAIL2"	Q 7.4	BOOL	//  (OA) - (FieldIO2-M4)
"PLRLL2"	Q 7.5	BOOL	//  (OA) - (FieldIO2-M4)
"SPI2"	Q 7.6	BOOL	//  (OA) - (FieldIO2-M4)
"TPFAIL2"	Q 7.7	BOOL	//  (OA) - (FieldIO2-M4)
"TM3"	Q 8.0	BOOL	//  (OPC) - (FieldIO3-M3)
"OPCO"	Q 8.1	BOOL	//  (OPC) - (FieldIO3-M3)
"SRVOLT"	Q 8.2	BOOL	//  (OPC) - (FieldIO3-M3)
"ASL"	Q 8.3	BOOL	//  (OPC) - (FieldIO3-M3)
"ASLDOR"	Q 8.4	BOOL	//  (OPC) - (FieldIO3-M3)
"CIV"	Q 8.5	BOOL	//  (OPC) - (FieldIO3-M3)
"EIVN"	Q 8.6	BOOL	//  (OPC) - (FieldIO3-M3)
"CIV1"	Q 8.7	BOOL	//  (OPC) - (FieldIO3-M3)
"CIV2"	Q 9.0	BOOL	//  (OPC) - (FieldIO3-M3)
"CIV3"	Q 9.1	BOOL	//  (OPC) - (FieldIO3-M3)
"CIV4"	Q 9.2	BOOL	//  (OPC) - (FieldIO3-M3)
"MSTPVL"	Q 9.3	BOOL	//  (OPC) - (FieldIO3-M3)
"MSTPVR"	Q 9.4	BOOL	//  (OPC) - (FieldIO3-M3)
"MTPRBMVP"	Q 9.5	BOOL	//  (OPC) - (FieldIO3-M3)
"TGRB"	Q 9.6	BOOL	//  (OPC) - (FieldIO3-M3)
"MANNAUTO"	Q 9.7	BOOL	//  (OA) - (FieldIO3-M3)
"HLLI"	Q 10.0	BOOL	//  (OA) - (FieldIO3-M4)
"LFRQO"	Q 10.1	BOOL	//  (OA) - (FieldIO3-M4)
"LLDO"	Q 10.2	BOOL	//  (OA) - (FieldIO3-M4)
"LLLI"	Q 10.3	BOOL	//  (OA) - (FieldIO3-M4)
"MOTO"	Q 10.4	BOOL	//  (OA) - (FieldIO3-M4)
"RBOP"	Q 10.5	BOOL	//  (OA) - (FieldIO3-M4)
"RCLINHO"	Q 10.6	BOOL	//  (OA) - (FieldIO3-M4)
"RCRINHO"	Q 10.7	BOOL	//  (OA) - (FieldIO3-M4)
"TSTRV1"	Q 11.0	BOOL	//  (OA) - (FieldIO3-M4)
"TSTRV2"	Q 11.1	BOOL	//  (OA) - (FieldIO3-M4)
"TSTRV3"	Q 11.2	BOOL	//  (OA) - (FieldIO3-M4)
"TSTRV4"	Q 11.3	BOOL	//  (OA) - (FieldIO3-M4)
"VPLL1"	Q 11.4	BOOL	//  (OA) - (FieldIO3-M4)
"VPLL2"	Q 11.5	BOOL	//  (OA) - (FieldIO3-M4)
"WSFAIL1"	Q 11.6	BOOL	//  (OA) - (FieldIO3-M4)
"WSFAIL2"	Q 11.7	BOOL	//  (OA) - (FieldIO3-M4)
"VAT (OPC-OA)"	VAT 1	
END_SYMBOL_TABLE

ORGANIZATION_BLOCK OB 1
TITLE = "Main Program Sweep (Cycle)"
VERSION : 0.1
VAR_TEMP
  OB1_EV_CLASS : BYTE ;	//Bits 0-3 = 1 (Coming event), Bits 4-7 = 1 (Event class 1)
  OB1_SCAN_1 : BYTE ;	//1 (Cold restart scan 1 of OB 1), 3 (Scan 2-n of OB 1)
  OB1_PRIORITY : BYTE ;	//Priority of OB Execution
  OB1_OB_NUMBR : BYTE ;	//1 (Organization block 1, OB1)
  OB1_RESERVED_1 : BYTE ;	//Reserved for system
  OB1_RESERVED_2 : BYTE ;	//Reserved for system
  OB1_PREV_CYCLE : INT ;	//Cycle time of previous OB1 scan (milliseconds)
  OB1_MIN_CYCLE : INT ;	//Minimum cycle time of OB1 (milliseconds)
  OB1_MAX_CYCLE : INT ;	//Maximum cycle time of OB1 (milliseconds)
  OB1_DATE_TIME : DATE_AND_TIME ;	//Date and time OB1 started
END_VAR
BEGIN
NETWORK
TITLE =
END_ORGANIZATION_BLOCK

ORGANIZATION_BLOCK "OBNL_FLT"	// OB 85
TITLE = "Organization Block (OB) Not Loaded Fault"
VERSION : 0.1
VAR_TEMP
  OB85_EV_CLASS : BYTE ;	//16#35 Event class 3
  OB85_FLT_ID : BYTE ;	//16#XX, Fault identification code
  OB85_PRIORITY : BYTE ;	//Priority of OB Execution
  OB85_OB_NUMBR : BYTE ;	//85 (Organization block 85, OB85)
  OB85_RESERVED_1 : BYTE ;	//Reserved for system
  OB85_RESERVED_2 : BYTE ;	//Reserved for system
  OB85_RESERVED_3 : INT ;	//Reserved for system
  OB85_ERR_EV_CLASS : BYTE ;	//Class of event causing error
  OB85_ERR_EV_NUM : BYTE ;	//Number of event causing error
  OB85_OB_PRIOR : BYTE ;	//Priority of OB causing error
  OB85_OB_NUM : BYTE ;	//Number of OB causing error
  OB85_DATE_TIME : DATE_AND_TIME ;	//Date and time OB85 started
END_VAR
BEGIN
// (block stored without names or comments; labels and parameter names are numbered)
END_ORGANIZATION_BLOCK

ORGANIZATION_BLOCK "PROG_ERR"	// OB 121
TITLE = "Programming Error"
VERSION : 0.1
VAR_TEMP
  OB121_EV_CLASS : BYTE ;	//16#25, Event class 2, Entering event state, Internal fault event
  OB121_SW_FLT : BYTE ;	//16#XX Software programming fault
  OB121_PRIORITY : BYTE ;	//Priority of OB Execution
  OB121_OB_NUMBR : BYTE ;	//121 (Organization block 121, OB121)
  OB121_BLK_TYPE : BYTE ;	//16#88/8A/8B/8C/8E Type of block fault occured in
  OB121_RESERVED_1 : BYTE ;	//Reserved for system
  OB121_FLT_REG : WORD ;	//16#XX Specific register that caused fault
  OB121_BLK_NUM : WORD ;	//Number of block that programming fault occured in
  OB121_PRG_ADDR : WORD ;	//Address in block where programming fault occured
  OB121_DATE_TIME : DATE_AND_TIME ;	//Date and time OB121 started
END_VAR
BEGIN
// (block stored without names or comments; labels and parameter names are numbered)
END_ORGANIZATION_BLOCK

ORGANIZATION_BLOCK "MOD_ERR"	// OB 122
TITLE = "Module Access Error"
VERSION : 0.1
VAR_TEMP
  OB122_EV_CLASS : BYTE ;	//16#29, Event class 2, Entering event state, Internal fault event
  OB122_SW_FLT : BYTE ;	//16#XX Software error code
  OB122_PRIORITY : BYTE ;	//Priority of OB Execution
  OB122_OB_NUMBR : BYTE ;	//122 (Organization block 122, OB122)
  OB122_BLK_TYPE : BYTE ;	//16#88/8C/8E Type of block fault occured in
  OB122_MEM_AREA : BYTE ;	//Memory area where access error occured
  OB122_MEM_ADDR : WORD ;	//Memory address where access error occured
  OB122_BLK_NUM : WORD ;	//Block number in which error occured
  OB122_PRG_ADDR : WORD ;	//Program address where error occured
  OB122_DATE_TIME : DATE_AND_TIME ;	//Date and time OB1 started
END_VAR
BEGIN
// (block stored without names or comments; labels and parameter names are numbered)
END_ORGANIZATION_BLOCK

